FUNCTION "Cage 12 unit" : VOID	// FC 25
TITLE = CAGE 12 UNIT FUNCTION
AUTHOR : Milesi
VERSION : 0.1
VAR_TEMP
  Brake_value : INT ;
END_VAR
BEGIN
NETWORK
TITLE = CAGE 12 OFF
      A(;
      L     "Cage 12".DB25_DBW2;
      L     0;
      ==I;
      );
      AN    "M180.1";
      AN    "M20.0";
      JNB   M001;
      R     "M188.0";
M001: NOP   0;
NETWORK
TITLE = CAGE 12 ON
      A(;
      L     "Cage 12".DB25_DBW2;
      L     1;
      ==I;
      );
      AN    "M180.1";
      AN    "M20.0";
      JNB   M002;
      S     "M188.0";
M002: NOP   0;
NETWORK
TITLE = CAGE 12 Z ROTATION
      A(;
      L     "Cage 12".DB25_DBW4;
      L     0;
      ==I;
      );
      AN    "M180.1";
      AN    "M20.0";
      JNB   M003;
      S     "M188.2";
      R     "M188.3";
M003: NOP   0;
NETWORK
TITLE = CAGE 12 S ROTATION
      A(;
      L     "Cage 12".DB25_DBW4;
      L     1;
      ==I;
      );
      AN    "M180.1";
      AN    "M20.0";
      JNB   M004;
      S     "M188.3";
      R     "M188.2";
M004: NOP   0;
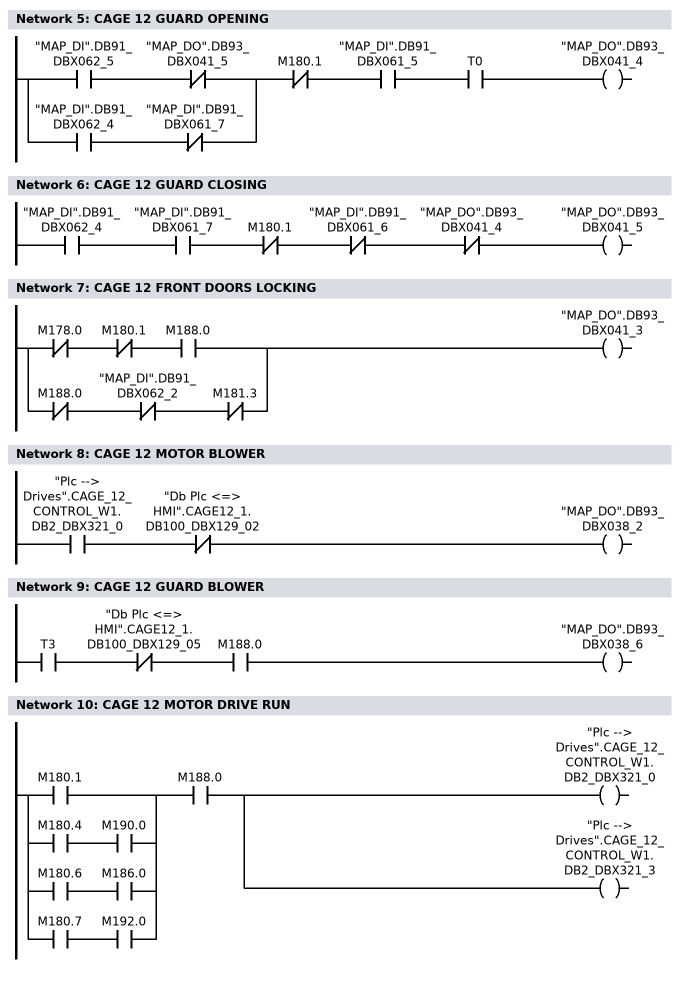
NETWORK
TITLE = CAGE 12 GUARD OPENING
      A(;
      A     "MAP_DI".DB91_DBX062_5;
      AN    "MAP_DO".DB93_DBX041_5;
      O;
      A     "MAP_DI".DB91_DBX062_4;
      AN    "MAP_DI".DB91_DBX061_7;
      );
      AN    "M180.1";
      A     "MAP_DI".DB91_DBX061_5;
      A     "T0";
      =     "MAP_DO".DB93_DBX041_4;
NETWORK
TITLE = CAGE 12 GUARD CLOSING
      A     "MAP_DI".DB91_DBX062_4;
      A     "MAP_DI".DB91_DBX061_7;
//      U     E     66.0
      AN    "M180.1";
      AN    "MAP_DI".DB91_DBX061_6;
      AN    "MAP_DO".DB93_DBX041_4;
      =     "MAP_DO".DB93_DBX041_5;
NETWORK
TITLE = CAGE 12 FRONT DOORS LOCKING
      AN    "M178.0";
      AN    "M180.1";
      A     "M188.0";
      O;
      AN    "M188.0";
      AN    "MAP_DI".DB91_DBX062_2;
      AN    "M181.3";
      =     "MAP_DO".DB93_DBX041_3;
NETWORK
TITLE = CAGE 12 MOTOR BLOWER 
      A     "Plc --> Drives".CAGE_12_CONTROL_W1.DB2_DBX321_0;
      AN    "Db Plc <=> HMI".CAGE12_1.DB100_DBX129_02;
      =     "MAP_DO".DB93_DBX038_2;
NETWORK
TITLE = CAGE 12 GUARD BLOWER
      A     "T3";
      AN    "Db Plc <=> HMI".CAGE12_1.DB100_DBX129_05;
      A     "M188.0";
      =     "MAP_DO".DB93_DBX038_6;
NETWORK
TITLE = CAGE 12 MOTOR DRIVE RUN
      A(;
      O     "M180.1";
      O;
      A     "M180.4";
      A     "M190.0";
      O;
      A     "M180.6";
      A     "M186.0";
      O;
      A     "M180.7";
      A     "M192.0";
      );
      A     "M188.0";
      =     "Plc --> Drives".CAGE_12_CONTROL_W1.DB2_DBX321_0;
      =     "Plc --> Drives".CAGE_12_CONTROL_W1.DB2_DBX321_3;
NETWORK
TITLE = CAGE 12 LAY SET ENABLE
      O     "M180.1";
      O     "M180.5";
      O(;
      A     "M180.4";
      A     "M190.0";
      );
      O(;
      A     "M180.6";
      A     "M186.0";
      );
      O(;
      A     "M180.7";
      A     "M192.0";
      );
      JC    M008;
      L     "Cage 12".DB25_DBD20;
      T     "Cage 12".DB25_DBD24;
      JU    M009;
M008: L     "Cage 12".DB25_DBD24;
      T     "Cage 12".DB25_DBD20;
M009: NOP   0;
NETWORK
TITLE = CAGE 12 MOTOR REFERENCE
//Max Linear Speed = 60 m/min
//Max Cage Rpm = 320
//
//Max Linear Speed              60000
//---------------- = Cage Lay = ----- = 187.5
//  Max Cage Rpm                 320
//
//                             Max Linear Speed
//Max Cage Rpm = 320 = 16384 = ---------------- * K
//                                Cage Lay
//
//    Cage Lay * 16384   187.5 * 16384
//K = ---------------- = ------------- = 51200
//    Max Linear Speed        60
// (network holds code this reader does not know; not shown)
//L     1.121200e+000
NETWORK
TITLE = CAGE 12 MAX LINEAR SPEED TO START
      AN    "M200.1";
      JNB   M00a;
      L     "Cage 12".DB25_DBD24;
      L     2.000000e-01;
      *R;
      JU    M00b;
M00a: L     "Cage 12".DB25_DBD24;
      L     2.600000e-01;
      *R;
M00b: T     "Cage 12".DB25_DBD120;
      O(;
      L     6.000000e+01;
      >R;
      );
      ON    "M188.0";
      JNB   M00c;
      T     "Cage 12".DB25_DBD120;
M00c: NOP   0;
NETWORK
TITLE = CAGE 12 MAX LINEAR SPEED
      L     "Cage 12".DB25_DBD24;
      L     3.200000e-01;
      *R;
      T     "Cage 12".DB25_DBD96;
      O(;
      L     6.000000e+01;
      >R;
      );
      ON    "M188.0";
      JNB   M00d;
      T     "Cage 12".DB25_DBD96;
M00d: NOP   0;
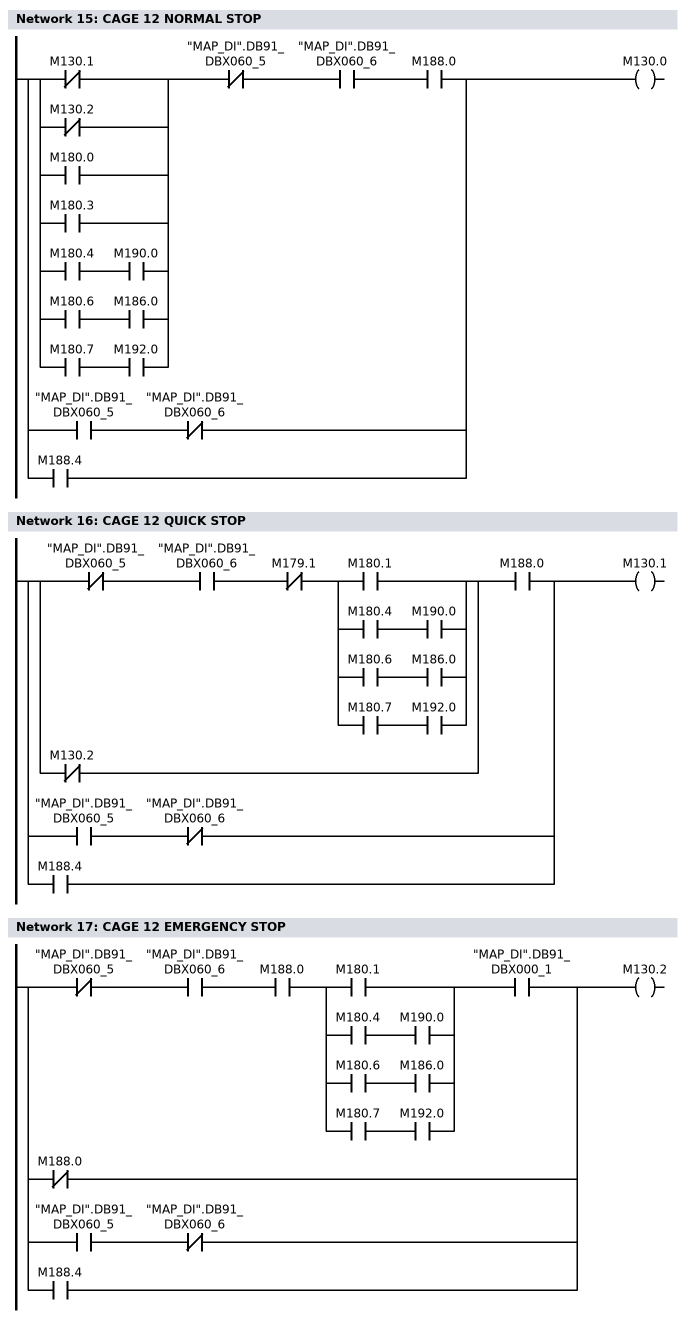
NETWORK
TITLE = CAGE 12 NORMAL STOP
      A(;
      ON    "M130.1";
      ON    "M130.2";
      O     "M180.0";
      O     "M180.3";
      O;
      A     "M180.4";
      A     "M190.0";
      O;
      A     "M180.6";
      A     "M186.0";
      O;
      A     "M180.7";
      A     "M192.0";
      );
      AN    "MAP_DI".DB91_DBX060_5;
      A     "MAP_DI".DB91_DBX060_6;
      A     "M188.0";
      O;
      A     "MAP_DI".DB91_DBX060_5;
      AN    "MAP_DI".DB91_DBX060_6;
      O     "M188.4";
      =     "M130.0";
NETWORK
TITLE = CAGE 12 QUICK STOP
      A(;
      AN    "MAP_DI".DB91_DBX060_5;
      A     "MAP_DI".DB91_DBX060_6;
      AN    "M179.1";
      A(;
      O     "M180.1";
      O;
      A     "M180.4";
      A     "M190.0";
      O;
      A     "M180.6";
      A     "M186.0";
      O;
      A     "M180.7";
      A     "M192.0";
      );
      ON    "M130.2";
      );
      A     "M188.0";
      O;
      A     "MAP_DI".DB91_DBX060_5;
      AN    "MAP_DI".DB91_DBX060_6;
      O     "M188.4";
      =     "M130.1";
NETWORK
TITLE = CAGE 12 EMERGENCY STOP
      AN    "MAP_DI".DB91_DBX060_5;
      A     "MAP_DI".DB91_DBX060_6;
      A     "M188.0";
      A(;
      O     "M180.1";
      O;
      A     "M180.4";
      A     "M190.0";
      O;
      A     "M180.6";
      A     "M186.0";
      O;
      A     "M180.7";
      A     "M192.0";
      );
      A     "MAP_DI".DB91_DBX000_1;
      ON    "M188.0";
      O;
      A     "MAP_DI".DB91_DBX060_5;
      AN    "MAP_DI".DB91_DBX060_6;
      O     "M188.4";
      =     "M130.2";
NETWORK
TITLE = CAGE 12 BRAKE PROPORTIONAL VALVE REFERENCE
      A     "M130.0";
      JC    M005;
      L     "Cage 12".DB25_DBD64;
      L     1.000000e+02;
      /R;
      L     2.764800e+04;
      *R;
      RND;
      JU    M006;
M005: A     "M130.1";
      JC    M007;
      L     "Cage 12".DB25_DBD68;
      L     1.000000e+02;
      /R;
      L     2.764800e+04;
      *R;
      RND;
      JU    M006;
M007: A     "M130.2";
      JC    M011;
      L     "Cage 12".DB25_DBD72;
      L     1.000000e+02;
      /R;
      L     2.764800e+04;
      *R;
      RND;
      JU    M006;
M011: L     0;
M006: T     #Brake_value;
NETWORK
TITLE = SET POINT IN AMPER CALCULATION
      L     "Cage 12".DB20_DBD276;
      L     1.360000e+02;
      *R;
      L     1.000000e+02;
      /R;
      T     "Cage 12".DB20_DBD260;
NETWORK
TITLE = CURRENT CALCULATION
// (network holds code this reader does not know; not shown)
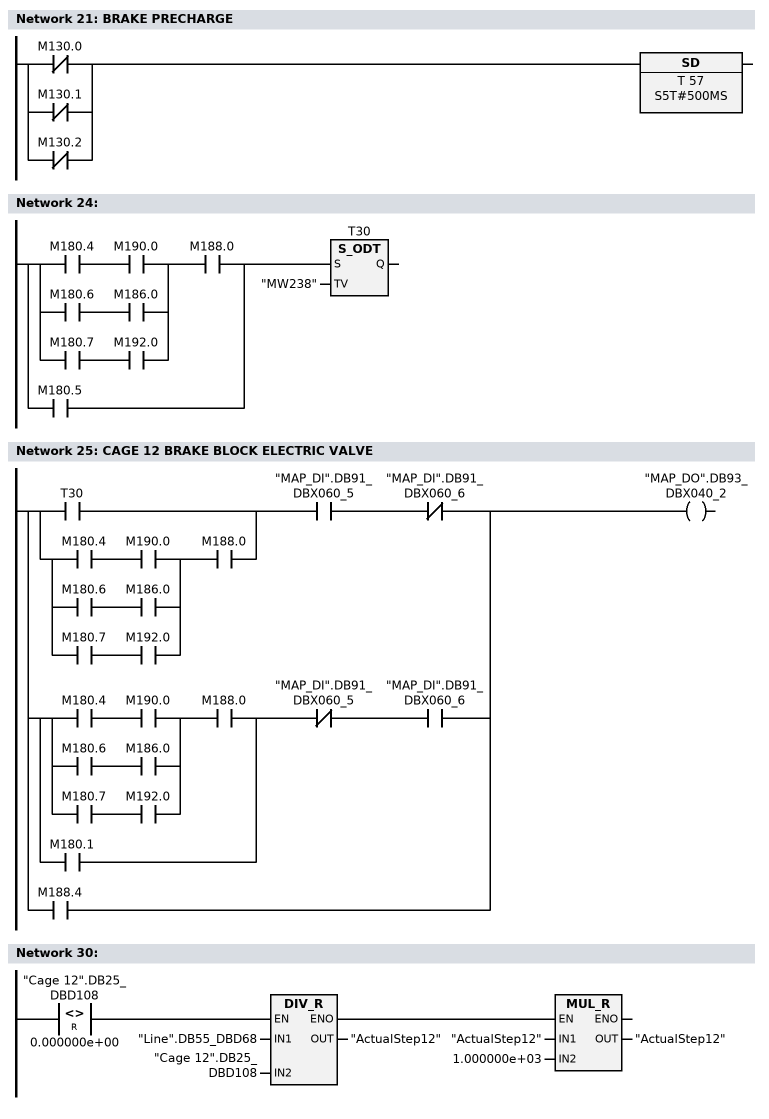
NETWORK
TITLE = BRAKE PRECHARGE
      ON    "M130.0";
      ON    "M130.1";
      ON    "M130.2";
      L     S5T#500MS;
      SD    T 57;
NETWORK
TITLE = BRAKE MODULATION CONTROL
      L     "Cage 12".DB20_DBD260;
      L     "Cage 12".DB25_DBD200;
      -R;
      T     "Cage 12".DB20_DBD264;
      L     "Cage 12".DB20_DBD268;
      *R;
      T     "Cage 12".DB20_DBD272;
      L     2.768400e+04;
      >R;
      JCN   M015;
      L     2.768400e+04;
      T     "Cage 12".DB20_DBD272;
M015: A     T 57;
      A     "M180.1";
      JCN   M016;
      A(;
      L     "Cage 12".DB20_DBD272;
      L     0.000000e+00;
      <R;
      );
      JCN   M017;
      L     0.000000e+00;
      T     "Cage 12".DB20_DBD272;
M017: L     "Cage 12".DB20_DBD272;
      RND;
      JU    M018;
M016: L     #Brake_value;
M018: T     "PAW286";
NETWORK
TITLE = CAGE 12 BRAKE BLOCK OPEN ON-DELAY TIMER
      L     "Cage 12".DB25_DBD148;
      RND;
      ITB;
      L     W#16#2000;
      OW;
      T     "MW238";
NETWORK
TITLE =
      A(;
      A(;
      A     "M180.4";
      A     "M190.0";
      O;
      A     "M180.6";
      A     "M186.0";
      O;
      A     "M180.7";
      A     "M192.0";
      );
      A     "M188.0";
      O     "M180.5";
      );
      L     "MW238";
      SD    "T30";
      NOP   0;
      NOP   0;
      NOP   0;
      NOP   0;
NETWORK
TITLE = CAGE 12 BRAKE BLOCK ELECTRIC VALVE
      A(;
      O     "T30";
      O;
      A(;
      O;
      A     "M180.4";
      A     "M190.0";
      O;
      A     "M180.6";
      A     "M186.0";
      O;
      A     "M180.7";
      A     "M192.0";
      );
      A     "M188.0";
      );
      A     "MAP_DI".DB91_DBX060_5;
      AN    "MAP_DI".DB91_DBX060_6;
      O;
      A(;
      A(;
      O;
      A     "M180.4";
      A     "M190.0";
      O;
      A     "M180.6";
      A     "M186.0";
      O;
      A     "M180.7";
      A     "M192.0";
      );
      A     "M188.0";
      O     "M180.1";
      );
      AN    "MAP_DI".DB91_DBX060_5;
      A     "MAP_DI".DB91_DBX060_6;
      O     "M188.4";
      =     "MAP_DO".DB93_DBX040_2;
NETWORK
TITLE = CAGE 12 RPM TO HMI
      L     "Drives --> Plc".DB1_DBW326;
      ITD;
      DTR;
      L     1.638400e+04;
      /R;
      L     3.200000e+02;
      *R;
      ABS;
      T     "Cage 12".DB25_DBD108;
NETWORK
TITLE = CAGE 12 MOTOR RPM TO HMI
      L     "Drives --> Plc".DB1_DBW326;
      ITD;
      DTR;
      L     1.638400e+04;
      /R;
      L     1.495000e+03;
      *R;
      T     "Cage 12".DB25_DBD188;
NETWORK
TITLE = CAGE 12 MOTOR CURRENT TO HMI
      L     "Drives --> Plc".DB1_DBW328;
      ITD;
      DTR;
      L     1.638400e+04;
      /R;
      L     1.360000e+02;
      *R;
      T     "Cage 12".DB25_DBD192;
NETWORK
TITLE = CAGE 12 MOTOR VOLTAGE TO HMI
      L     "Drives --> Plc".DB1_DBW330;
      ITD;
      DTR;
      L     1.638400e+04;
      /R;
      L     4.000000e+02;
      *R;
      T     "Cage 12".DB25_DBD196;
NETWORK
TITLE =
      A(;
      A(;
      L     "Cage 12".DB25_DBD108;
      L     0.000000e+00;
      <>R;
      );
      JNB   _001;
      L     "Line".DB55_DBD68;
      L     "Cage 12".DB25_DBD108;
      /R;
      T     "ActualStep12";
      AN    OV;
      SAVE;
      CLR;
_001: A     BR;
      );
      JNB   _002;
      L     "ActualStep12";
      L     1.000000e+03;
      *R;
      T     "ActualStep12";
_002: NOP   0;
END_FUNCTION

FUNCTION "Cage 12 loading fase" : VOID	// FC 26
TITLE = CAGE 12 LOADING FASE FUNCTION
AUTHOR : Milesi
VERSION : 0.1
BEGIN
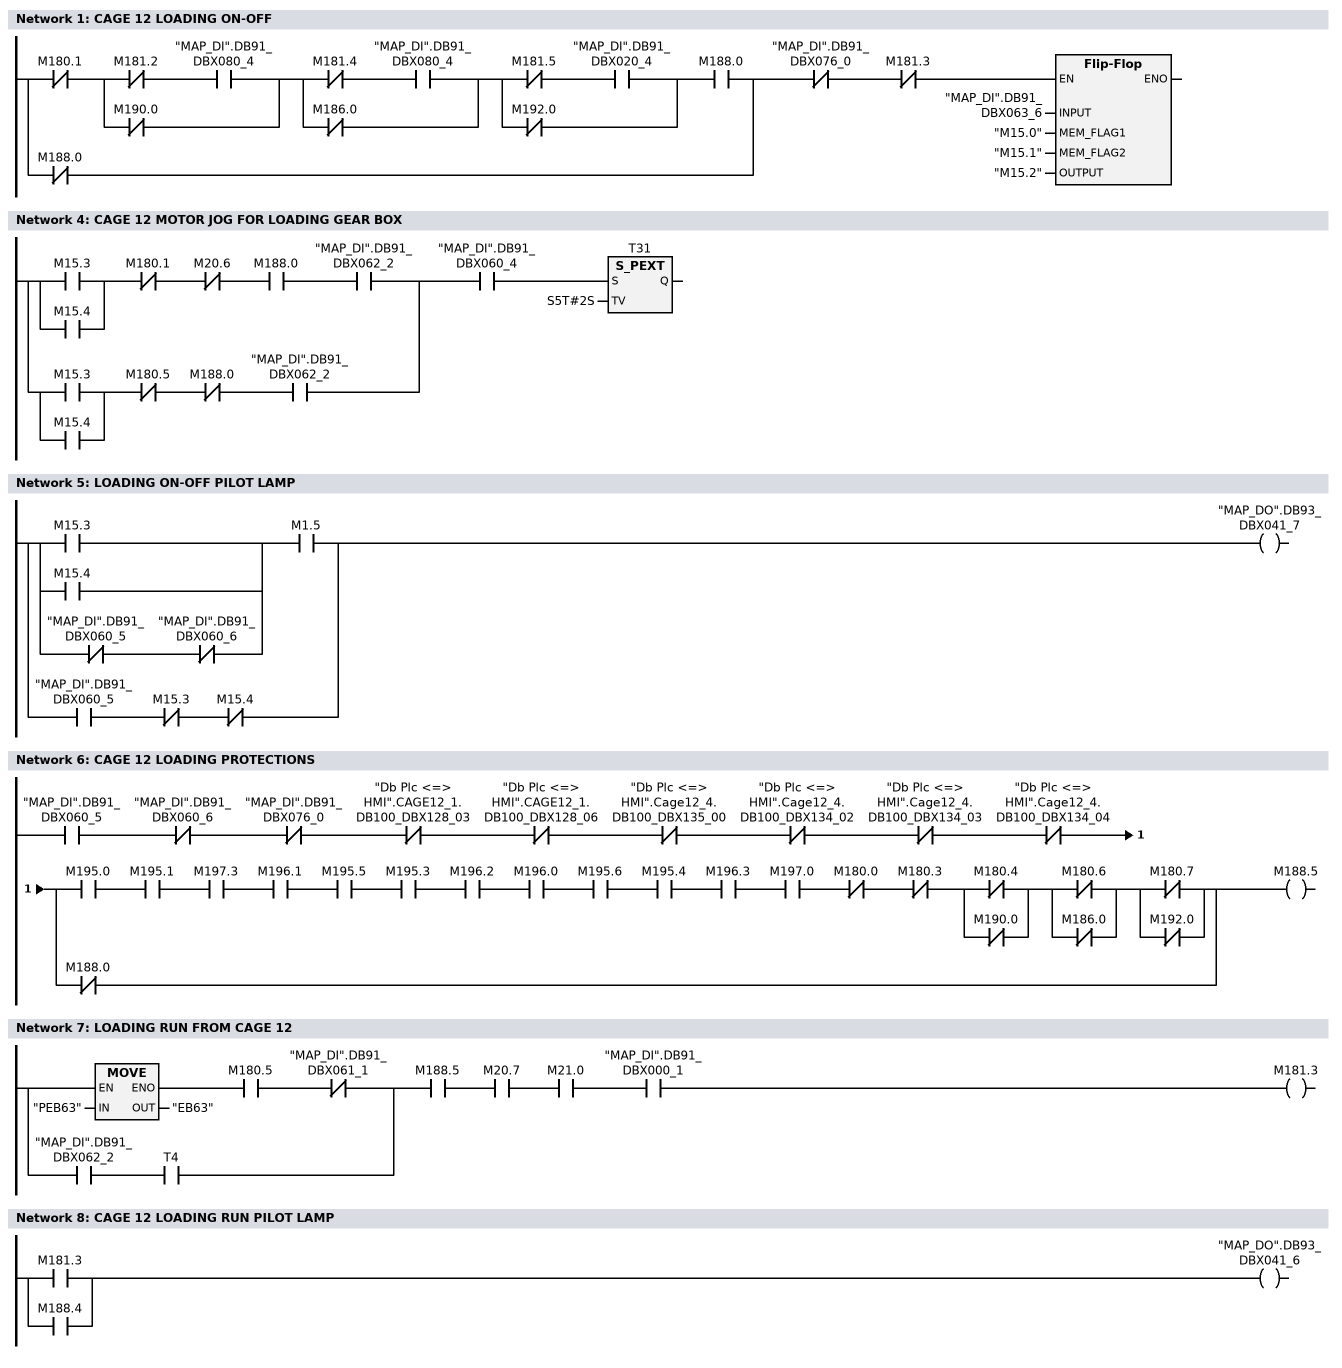
NETWORK
TITLE = CAGE 12 LOADING ON-OFF
      A(;
      AN    "M180.1";
      A(;
      AN    "M181.2";
      A     "MAP_DI".DB91_DBX080_4;
      ON    "M190.0";
      );
      A(;
      AN    "M181.4";
      A     "MAP_DI".DB91_DBX080_4;
      ON    "M186.0";
      );
      A(;
      AN    "M181.5";
      A     "MAP_DI".DB91_DBX020_4;
      ON    "M192.0";
      );
      A     "M188.0";
      ON    "M188.0";
      );
      AN    "MAP_DI".DB91_DBX076_0;
      AN    "M181.3";
      JNB   _001;
      CALL  "Flip-Flop" (
           INPUT                    := "MAP_DI".DB91_DBX063_6,
           MEM_FLAG1                := "M15.0",
           MEM_FLAG2                := "M15.1",
           OUTPUT                   := "M15.2");
_001: NOP   0;
NETWORK
TITLE = CAGE 12 LOADING ON
      A(;
      A(;
      A     "M15.2";
      AN    "M180.1";
      AN    "M20.6";
      A     "M188.0";
      O;
      AN    "M180.5";
      AN    "M188.0";
      );
      S     "MAP_DO".DB93_DBX040_0;
      A(;
      O     "MAP_DI".DB91_DBX060_5;
      O     "MAP_DO".DB93_DBX040_1;
      ON    "M15.2";
      );
      R     "MAP_DO".DB93_DBX040_0;
      A     "MAP_DO".DB93_DBX040_0;
      );
      S     "M15.3";
      A(;
      O     "MAP_DI".DB91_DBX060_5;
      ON    "M15.2";
      );
      R     "M15.3";
      NOP   0;
NETWORK
TITLE = CAGE 12 LOADING OFF
      A(;
      A(;
      AN    "M15.2";
      AN    "M20.6";
      A     "M188.0";
      O;
      AN    "M180.5";
      AN    "M188.0";
      );
      S     "MAP_DO".DB93_DBX040_1;
      A(;
      O     "MAP_DI".DB91_DBX060_6;
      O     "MAP_DO".DB93_DBX040_0;
      O     "M15.2";
      );
      R     "MAP_DO".DB93_DBX040_1;
      A     "MAP_DO".DB93_DBX040_1;
      );
      S     "M15.4";
      A(;
      O     "MAP_DI".DB91_DBX060_6;
      O     "M15.2";
      );
      R     "M15.4";
      NOP   0;
NETWORK
TITLE = CAGE 12 MOTOR JOG FOR LOADING GEAR BOX
      A(;
      A(;
      O     "M15.3";
      O     "M15.4";
      );
      AN    "M180.1";
      AN    "M20.6";
      A     "M188.0";
      A     "MAP_DI".DB91_DBX062_2;
      O;
      A(;
      O     "M15.3";
      O     "M15.4";
      );
      AN    "M180.5";
      AN    "M188.0";
      A     "MAP_DI".DB91_DBX062_2;
      );
      A     "MAP_DI".DB91_DBX060_4;
      L     S5T#2S;
      SE    "T31";
      NOP   0;
      NOP   0;
      NOP   0;
      NOP   0;
NETWORK
TITLE = LOADING ON-OFF PILOT LAMP
      A(;
      O     "M15.3";
      O     "M15.4";
      O;
      AN    "MAP_DI".DB91_DBX060_5;
      AN    "MAP_DI".DB91_DBX060_6;
      );
      A     "M1.5";
      O;
      A     "MAP_DI".DB91_DBX060_5;
      AN    "M15.3";
      AN    "M15.4";
      =     "MAP_DO".DB93_DBX041_7;
NETWORK
TITLE = CAGE 12 LOADING PROTECTIONS
      A     "MAP_DI".DB91_DBX060_5;
      AN    "MAP_DI".DB91_DBX060_6;
      AN    "MAP_DI".DB91_DBX076_0;
      AN    "Db Plc <=> HMI".CAGE12_1.DB100_DBX128_03;
      AN    "Db Plc <=> HMI".CAGE12_1.DB100_DBX128_06;
      AN    "Db Plc <=> HMI".Cage12_4.DB100_DBX135_00;
      AN    "Db Plc <=> HMI".Cage12_4.DB100_DBX134_02;
      AN    "Db Plc <=> HMI".Cage12_4.DB100_DBX134_03;
      AN    "Db Plc <=> HMI".Cage12_4.DB100_DBX134_04;
      A(;
      A     "M195.0";
      A     "M195.1";
      A     "M197.3";
      A     "M196.1";
      A     "M195.5";
      A     "M195.3";
      A     "M196.2";
      A     "M196.0";
      A     "M195.6";
      A     "M195.4";
      A     "M196.3";
      A     "M197.0";
      AN    "M180.0";
      AN    "M180.3";
      A(;
      ON    "M180.4";
      ON    "M190.0";
      );
      A(;
      ON    "M180.6";
      ON    "M186.0";
      );
      A(;
      ON    "M180.7";
      ON    "M192.0";
      );
      ON    "M188.0";
      );
      =     "M188.5";
NETWORK
TITLE = LOADING RUN FROM CAGE 12
      A(;
      A(;
      L     "PEB63";
      T     "EB63";
      SET;
      SAVE;
      CLR;
      A     BR;
      );
      A     "M180.5";
      AN    "MAP_DI".DB91_DBX061_1;
      O;
      A     "MAP_DI".DB91_DBX062_2;
      A     "T4";
      );
      A     "M188.5";
      A     "M20.7";
      A     "M21.0";
      A     "MAP_DI".DB91_DBX000_1;
      =     "M181.3";
NETWORK
TITLE = CAGE 12 LOADING RUN PILOT LAMP
      O     "M181.3";
      O     "M188.4";
      =     "MAP_DO".DB93_DBX041_6;
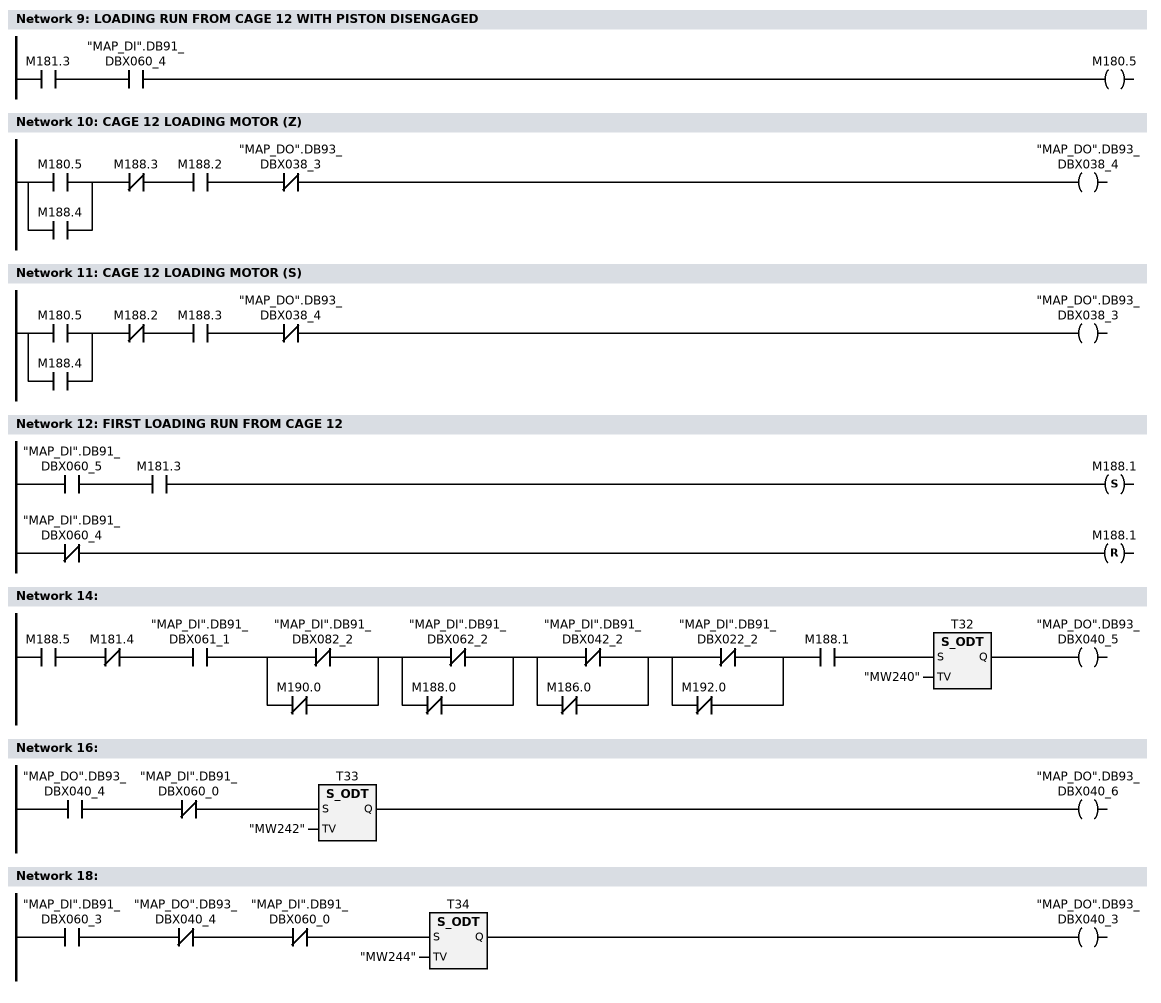
NETWORK
TITLE = LOADING RUN FROM CAGE 12 WITH PISTON DISENGAGED
      A     "M181.3";
      A     "MAP_DI".DB91_DBX060_4;
      =     "M180.5";
NETWORK
TITLE = CAGE 12 LOADING MOTOR (Z)
      A(;
      O     "M180.5";
      O     "M188.4";
      );
      AN    "M188.3";
      A     "M188.2";
      AN    "MAP_DO".DB93_DBX038_3;
      =     "MAP_DO".DB93_DBX038_4;
NETWORK
TITLE = CAGE 12 LOADING MOTOR (S)
      A(;
      O     "M180.5";
      O     "M188.4";
      );
      AN    "M188.2";
      A     "M188.3";
      AN    "MAP_DO".DB93_DBX038_4;
      =     "MAP_DO".DB93_DBX038_3;
NETWORK
TITLE = FIRST LOADING RUN FROM CAGE 12
      A     "MAP_DI".DB91_DBX060_5;
      A     "M181.3";
      S     "M188.1";
      AN    "MAP_DI".DB91_DBX060_4;
      R     "M188.1";
      NOP   0;
NETWORK
TITLE = CAGE 12 PISTON ENGAGING INTO CAGE
      L     "Cage 12".DB25_DBD152;
      RND;
      ITB;
      L     W#16#2000;
      OW;
      T     "MW240";
NETWORK
TITLE =
      A     "M188.5";
      AN    "M181.4";
      A     "MAP_DI".DB91_DBX061_1;
      A(;
      ON    "MAP_DI".DB91_DBX082_2;
      ON    "M190.0";
      );
      A(;
      ON    "MAP_DI".DB91_DBX062_2;
      ON    "M188.0";
      );
      A(;
      ON    "MAP_DI".DB91_DBX042_2;
      ON    "M186.0";
      );
      A(;
      ON    "MAP_DI".DB91_DBX022_2;
      ON    "M192.0";
      );
      A     "M188.1";
      L     "MW240";
      SD    "T32";
      NOP   0;
      NOP   0;
      NOP   0;
      A     "T32";
      =     "MAP_DO".DB93_DBX040_5;
NETWORK
TITLE = CAGE 12 PISTON DISENGAGING FROM CAGE
      L     "Cage 12".DB25_DBD144;
      RND;
      ITB;
      L     W#16#2000;
      OW;
      T     "MW242";
NETWORK
TITLE =
      A     "MAP_DO".DB93_DBX040_4;
      AN    "MAP_DI".DB91_DBX060_0;
      L     "MW242";
      SD    "T33";
      NOP   0;
      NOP   0;
      NOP   0;
      A     "T33";
      =     "MAP_DO".DB93_DBX040_6;
NETWORK
TITLE = CAGE 12 AIR INLET INTO CAGE
      L     "Cage 12".DB25_DBD156;
      RND;
      ITB;
      L     W#16#2000;
      OW;
      T     "MW244";
NETWORK
TITLE =
      A     "MAP_DI".DB91_DBX060_3;
      AN    "MAP_DO".DB93_DBX040_4;
      AN    "MAP_DI".DB91_DBX060_0;
      L     "MW244";
      SD    "T34";
      NOP   0;
      NOP   0;
      NOP   0;
      A     "T34";
      =     "MAP_DO".DB93_DBX040_3;
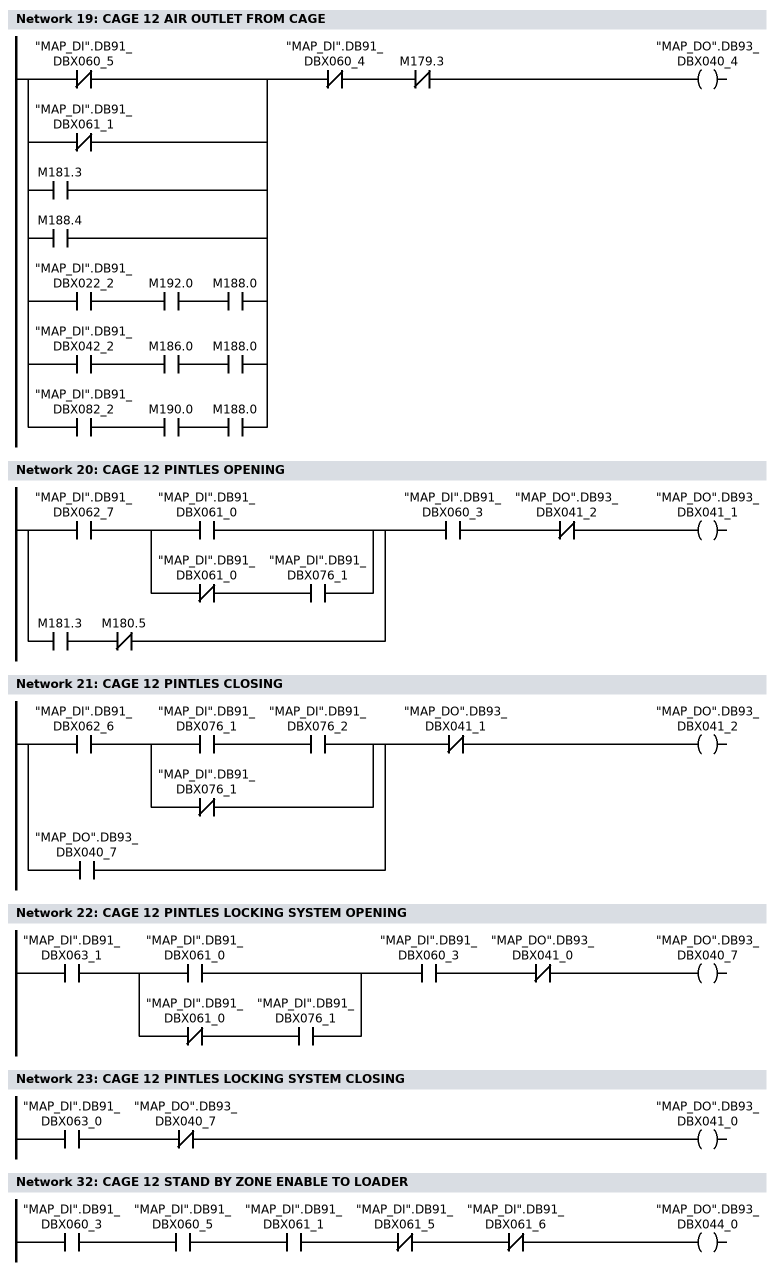
NETWORK
TITLE = CAGE 12 AIR OUTLET FROM CAGE
      A(;
      ON    "MAP_DI".DB91_DBX060_5;
      ON    "MAP_DI".DB91_DBX061_1;
      O     "M181.3";
      O     "M188.4";
      O;
      A     "MAP_DI".DB91_DBX022_2;
      A     "M192.0";
      A     "M188.0";
      O;
      A     "MAP_DI".DB91_DBX042_2;
      A     "M186.0";
      A     "M188.0";
      O;
      A     "MAP_DI".DB91_DBX082_2;
      A     "M190.0";
      A     "M188.0";
      );
      AN    "MAP_DI".DB91_DBX060_4;
      AN    "M179.3";
      =     "MAP_DO".DB93_DBX040_4;
NETWORK
TITLE = CAGE 12 PINTLES OPENING
      A(;
      A     "MAP_DI".DB91_DBX062_7;
      A(;
      O     "MAP_DI".DB91_DBX061_0;
      O;
      AN    "MAP_DI".DB91_DBX061_0;
      A     "MAP_DI".DB91_DBX076_1;
      );
      O;
      A     "M181.3";
      AN    "M180.5";
      );
      A     "MAP_DI".DB91_DBX060_3;
      AN    "MAP_DO".DB93_DBX041_2;
      =     "MAP_DO".DB93_DBX041_1;
NETWORK
TITLE = CAGE 12 PINTLES CLOSING
      A(;
      A     "MAP_DI".DB91_DBX062_6;
      A(;
      A     "MAP_DI".DB91_DBX076_1;
      A     "MAP_DI".DB91_DBX076_2;
      ON    "MAP_DI".DB91_DBX076_1;
      );
      O     "MAP_DO".DB93_DBX040_7;
      );
      AN    "MAP_DO".DB93_DBX041_1;
      =     "MAP_DO".DB93_DBX041_2;
NETWORK
TITLE = CAGE 12 PINTLES LOCKING SYSTEM OPENING
      A     "MAP_DI".DB91_DBX063_1;
      A(;
      O     "MAP_DI".DB91_DBX061_0;
      O;
      AN    "MAP_DI".DB91_DBX061_0;
      A     "MAP_DI".DB91_DBX076_1;
      );
      A     "MAP_DI".DB91_DBX060_3;
      AN    "MAP_DO".DB93_DBX041_0;
      =     "MAP_DO".DB93_DBX040_7;
NETWORK
TITLE = CAGE 12 PINTLES LOCKING SYSTEM CLOSING
      A     "MAP_DI".DB91_DBX063_0;
      AN    "MAP_DO".DB93_DBX040_7;
      =     "MAP_DO".DB93_DBX041_0;
NETWORK
TITLE = CAGE 12 PLATFORM UP
NETWORK
TITLE = CAGE 12 PLATFORM DOWN
NETWORK
TITLE = CAGE 12 EVEN BOBBINS ROTATION FOR LOADING MACHINE
NETWORK
TITLE = CAGE 12 EVEN BOBBINS ROTATION FOR LOADING PLATFORM
NETWORK
TITLE = CAGE 12 ODD BOBBINS ROTATION FOR LOADING MACHINE
NETWORK
TITLE = CAGE 12 ODD BOBBINS ROTATION FOR LOADING PLATFORM
NETWORK
TITLE = CAGE 12 BOBBIN ROTATION FOR LOADING MACHINE PILOT LAMP
NETWORK
TITLE = CAGE 12 LOADING PUMP
NETWORK
TITLE = CAGE 12 STAND BY ZONE ENABLE TO LOADER
      A     "MAP_DI".DB91_DBX060_3;
      A     "MAP_DI".DB91_DBX060_5;
      A     "MAP_DI".DB91_DBX061_1;
      AN    "MAP_DI".DB91_DBX061_5;
      AN    "MAP_DI".DB91_DBX061_6;
      =     "MAP_DO".DB93_DBX044_0;
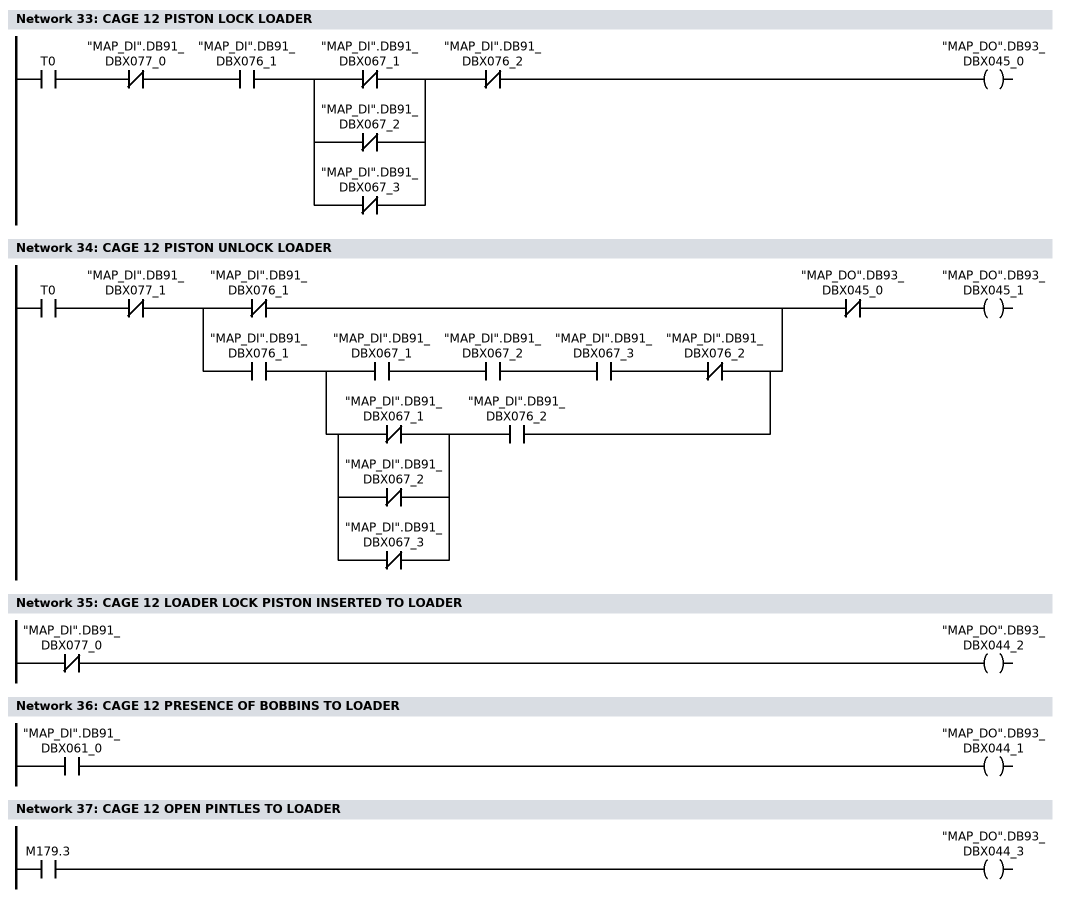
NETWORK
TITLE = CAGE 12 PISTON LOCK LOADER
      A     "T0";
      AN    "MAP_DI".DB91_DBX077_0;
      A     "MAP_DI".DB91_DBX076_1;
      A(;
      ON    "MAP_DI".DB91_DBX067_1;
      ON    "MAP_DI".DB91_DBX067_2;
      ON    "MAP_DI".DB91_DBX067_3;
      );
      AN    "MAP_DI".DB91_DBX076_2;
      =     "MAP_DO".DB93_DBX045_0;
NETWORK
TITLE = CAGE 12 PISTON UNLOCK LOADER
      A     "T0";
      AN    "MAP_DI".DB91_DBX077_1;
      A(;
      ON    "MAP_DI".DB91_DBX076_1;
      O;
      A     "MAP_DI".DB91_DBX076_1;
      A(;
      A     "MAP_DI".DB91_DBX067_1;
      A     "MAP_DI".DB91_DBX067_2;
      A     "MAP_DI".DB91_DBX067_3;
      AN    "MAP_DI".DB91_DBX076_2;
      O;
      A(;
      ON    "MAP_DI".DB91_DBX067_1;
      ON    "MAP_DI".DB91_DBX067_2;
      ON    "MAP_DI".DB91_DBX067_3;
      );
      A     "MAP_DI".DB91_DBX076_2;
      );
      );
      AN    "MAP_DO".DB93_DBX045_0;
      =     "MAP_DO".DB93_DBX045_1;
NETWORK
TITLE = CAGE 12 LOADER LOCK PISTON INSERTED TO LOADER 
      AN    "MAP_DI".DB91_DBX077_0;
      =     "MAP_DO".DB93_DBX044_2;
NETWORK
TITLE = CAGE 12 PRESENCE OF BOBBINS TO LOADER
      A     "MAP_DI".DB91_DBX061_0;
      =     "MAP_DO".DB93_DBX044_1;
NETWORK
TITLE = CAGE 12 OPEN PINTLES TO LOADER
      A     "M179.3";
      =     "MAP_DO".DB93_DBX044_3;
END_FUNCTION

FUNCTION "Cage 12 preforming alarm" : VOID	// FC 27
TITLE = CAGE 12 PREFORMING ALARMS FUNCTION
AUTHOR : Milesi
VERSION : 0.1
BEGIN
NETWORK
TITLE = CAGE 12 PREFORMING MOTOR DRIVE PROFIBUS SLAVE 10 FAULT
      A(;
      L     "MB304";
      L     10;
      ==I;
      );
      AN    "M300.5";
      S     "Db Plc <=> HMI".PROFIBUS.DB100_DBX100_1;
NETWORK
TITLE = CAGE 12 PREFORMING MOTOR BRAKE OVERLOAD
      A     "T0";
      A     "MAP_DI".DB91_DBX058_4;
      A     "M189.3";
      =     "Db Plc <=> HMI".Cage12_4.DB100_DBX135_04;
NETWORK
TITLE = CAGE 12 PREFORMING MOTOR BLOWER OVERLOAD
      A     "T0";
      A     "MAP_DI".DB91_DBX058_5;
      A     "M189.3";
      =     "Db Plc <=> HMI".Cage12_4.DB100_DBX135_05;
NETWORK
TITLE = CAGE 12 PREFORMING OPEN GUARD
      A     "T0";
      A     "M180.1";
      AN    "MAP_DI".DB91_DBX064_6;
      A     "M189.3";
      S     "M174.5";
NETWORK
TITLE =
      A     "T0";
      A(;
      ON    "MAP_DI".DB91_DBX064_6;
      O     "M174.5";
      );
      A     "M189.3";
      =     "Db Plc <=> HMI".Cage12_4.DB100_DBX135_06;
NETWORK
TITLE = CAGE 12 PREFORMING MOTOR DRIVE FAULT
      A     "T0";
      A     "Drives --> Plc".CAGE_12_PREF_STATUS_W1.DB1_DBX281_3;
      A     "M189.3";
      S     "Db Plc <=> HMI".Cage12_4.DB100_DBX135_07;
NETWORK
TITLE = CAGE 12 PREFORMING GENERAL ALARM
      AN    "Db Plc <=> HMI".PROFIBUS.DB100_DBX100_1;
      AN    "Db Plc <=> HMI".Cage12_4.DB100_DBX135_04;
      AN    "Db Plc <=> HMI".Cage12_4.DB100_DBX135_05;
      AN    "Db Plc <=> HMI".Cage12_4.DB100_DBX135_06;
      AN    "Db Plc <=> HMI".Cage12_4.DB100_DBX135_07;
      =     "M196.0";
END_FUNCTION

FUNCTION "Cage 12 preforming unit" : VOID	// FC 28
TITLE = CAGE 12 PREFORMING UNIT FUNCTION
AUTHOR : Milesi
VERSION : 0.1
BEGIN
NETWORK
TITLE = CAGE 12 PREFORMING OFF
      A(;
      L     "Cage 12 preforming".DB28_DBW2;
      L     0;
      ==I;
      );
      AN    "M180.1";
      JNB   _001;
      R     "M189.3";
      R     "M189.4";
      R     "M189.5";
_001: NOP   0;
NETWORK
TITLE = CAGE 12 PREFORMING Z ROTATION
      A(;
      L     "Cage 12 preforming".DB28_DBW2;
      L     1;
      ==I;
      );
      AN    "M180.1";
      JNB   _002;
      S     "M189.3";
      S     "M189.4";
      R     "M189.5";
_002: NOP   0;
NETWORK
TITLE = CAGE 12 PREFORMING S ROTATION
      A(;
      L     "Cage 12 preforming".DB28_DBW2;
      L     2;
      ==I;
      );
      AN    "M180.1";
      JNB   _003;
      S     "M189.3";
      S     "M189.5";
      R     "M189.4";
_003: NOP   0;
NETWORK
TITLE = CAGE 12 PREFORMING MOTOR DRIVE RUN
      A(;
      O     "M180.1";
      O     "M21.3";
      );
      AN    "Db Plc <=> HMI".Cage12_4.DB100_DBX135_07;
      A     "M189.3";
      =     "Plc --> Drives".CAGE_12_PREF_CONTROL_W1.DB2_DBX281_0;
      =     "Plc --> Drives".CAGE_12_PREF_CONTROL_W1.DB2_DBX281_3;
NETWORK
TITLE = CAGE 12 PREFORMING MOTOR BLOWER
      A     "Plc --> Drives".CAGE_12_PREF_CONTROL_W1.DB2_DBX281_0;
      AN    "Db Plc <=> HMI".Cage12_4.DB100_DBX135_05;
      =     "MAP_DO".DB93_DBX038_1;
NETWORK
TITLE = CAGE 12 PREFORMING MOTOR ELECTRIC BRAKE RELAY
      A(;
      O     "Plc --> Drives".CAGE_12_PREF_CONTROL_W1.DB2_DBX281_0;
      O     "MAP_DI".DB91_DBX064_7;
      );
      AN    "Db Plc <=> HMI".Cage12_4.DB100_DBX135_05;
      =     "MAP_DO".DB93_DBX038_0;
NETWORK
TITLE = CAGE 12 PREFORMING MOTOR REFERENCE
//Max Linear Speed = 40 m/min
//Max Die Rpm = 147.68
//
//Max Linear Speed             40000
//---------------- = Die Lay = ------ = 270.85
//  Max Die Rpm                147.68
//
//                               Max Linear Speed
//Max Die Rpm = 147.68 = 16384 = ---------------- * K
//                                   Die Lay
//
//    Die Lay * 16384   270.85 * 16384
//K = ---------------- = ------------- = 110940.16
//    Max Linear Speed        40
// (network holds code this reader does not know; not shown)
NETWORK
TITLE = CAGE 12 PREFORMING RPM TO HMI
      L     "Drives --> Plc".DB1_DBW286;
      ITD;
      DTR;
      L     1.638400e+04;
      /R;
      L     1.476800e+02;
      *R;
      ABS;
      T     "Cage 12 preforming".DB28_DBD108;
NETWORK
TITLE = CAGE 12 PREFORMING MOTOR RPM TO HMI
      L     "Drives --> Plc".DB1_DBW286;
      ITD;
      DTR;
      L     1.638400e+04;
      /R;
      L     1.420000e+03;
      *R;
      T     "Cage 12 preforming".DB28_DBD188;
NETWORK
TITLE = CAGE 12 PREFORMING MOTOR CURRENT TO HMI
//TORQUE FEEDBACK = 150% = MOTOR CURRENT * 1.5
      L     "Drives --> Plc".DB1_DBW288;
      ITD;
      DTR;
      L     1.638400e+04;
      /R;
      L     3.400000e+00;
      *R;
      T     "Cage 12 preforming".DB28_DBD192;
NETWORK
TITLE = CAGE 12 PREFORMING MOTOR VOLTAGE TO HMI
      L     "Drives --> Plc".DB1_DBW290;
      ITD;
      DTR;
      L     1.638400e+04;
      /R;
      L     4.000000e+02;
      *R;
      T     "Cage 12 preforming".DB28_DBD196;
END_FUNCTION

FUNCTION "Cage 6 alarms" : VOID	// FC 29
TITLE = CAGE 6 ALARMS FUNCTION
AUTHOR : Milesi
VERSION : 0.1
VAR_TEMP
  T4_time : WORD ;
END_VAR
BEGIN
NETWORK
TITLE = CAGE 6 MOTOR DRIVE PROFIBUS SLAVE 12 FAULT
      A(;
      L     "MB304";
      L     12;
      ==I;
      );
      AN    "M300.5";
      S     "Db Plc <=> HMI".PROFIBUS.DB100_DBX100_3;
NETWORK
TITLE = CAGE 6 ET200M PROFIBUS SLAVE 24 FAULT
      A(;
      L     "MB304";
      L     24;
      ==I;
      );
      AN    "M300.5";
      S     "Db Plc <=> HMI".PROFIBUS_1.DB100_DBX103_0;
NETWORK
TITLE = CAGE 6 OPEN FRONT GUARD
      A     "T0";
      A     "M180.1";
      AN    "MAP_DI".DB91_DBX081_6;
      A     "M190.0";
      S     "M173.1";
NETWORK
TITLE =
      A     "T0";
      A(;
      ON    "MAP_DI".DB91_DBX081_6;
      O     "M173.1";
      );
      A     "M190.0";
      =     "Db Plc <=> HMI".Cage6_1.DB100_DBX136_0;
NETWORK
TITLE = CAGE 6 PRESENCE OF MAN
      A     "T0";
      AN    "MAP_DI".DB91_DBX081_7;
      AN    "M180.1";
      A     "M190.0";
      =     "Db Plc <=> HMI".Cage6_1.DB100_DBX136_1;
NETWORK
TITLE = CAGE 6 LOADING ENGAGED
      A     "T0";
      A     "MAP_DI".DB91_DBX080_5;
      AN    "MAP_DI".DB91_DBX080_6;
      A     "M14.2";
      =     "Db Plc <=> HMI".Cage6_1.DB100_DBX136_2;
NETWORK
TITLE = CAGE 6 LOADING GEAR BOX NOT ENGAGED
      A     "T0";
      AN    "MAP_DI".DB91_DBX080_5;
      AN    "MAP_DI".DB91_DBX080_6;
      =     "Db Plc <=> HMI".Cage6_1.DB100_DBX136_3;
NETWORK
TITLE = CAGE 6 LOADING MOTOR OVERLOAD
      A     "T0";
      A     "MAP_DI".DB91_DBX078_4;
      =     "Db Plc <=> HMI".Cage6_1.DB100_DBX136_6;
NETWORK
TITLE = CAGE 6 AIR PIPE NOT IN POSITION
      A     "T0";
      A     "M180.1";
      AN    "MAP_DI".DB91_DBX080_7;
      A     "M190.0";
      S     "M173.2";
NETWORK
TITLE =
      A     "T0";
      A(;
      ON    "MAP_DI".DB91_DBX080_7;
      O     "M173.2";
      );
      =     "Db Plc <=> HMI".Cage6_1.DB100_DBX136_5;
NETWORK
TITLE = CAGE 6 PISTON INSIDE CAGE
      A     "T0";
      A     "M180.1";
      AN    "MAP_DI".DB91_DBX080_4;
      A     "M190.0";
      S     "M171.5";
NETWORK
TITLE =
      A     "T0";
      A(;
      ON    "MAP_DI".DB91_DBX080_4;
      O     "M171.5";
      );
      =     "Db Plc <=> HMI".Cage6_1.DB100_DBX136_7;
NETWORK
TITLE = CAGE 6 24VDC POWER SUPPLY OVERLOAD
      A     "T0";
      AN    "MAP_DI".DB91_DBX078_3;
      =     "Db Plc <=> HMI".Cage6_1.DB100_DBX137_0;
NETWORK
TITLE = CAGE 6 220VAC POWER SUPPLY OVERLOAD
      A     "T0";
      AN    "MAP_DI".DB91_DBX078_2;
      =     "Db Plc <=> HMI".Cage6_1.DB100_DBX137_1;
NETWORK
TITLE = CAGE 6 MOTOR BLOWER OVERLOAD
      A     "T0";
      A     "MAP_DI".DB91_DBX078_5;
      =     "Db Plc <=> HMI".Cage6_1.DB100_DBX137_2;
NETWORK
TITLE = CAGE 6 LOADING PLATFORM MOTOR OVERLOAD
NETWORK
TITLE = CAGE 6 GUARD BLOWER MOTOR OVERLOAD
      A     "T0";
      A     "MAP_DI".DB91_DBX078_7;
      =     "Db Plc <=> HMI".Cage6_1.DB100_DBX137_5;
NETWORK
TITLE = CAGE 6 OPEN FRONT DOOR
//      U(    
//      U(    
//      U     T      0
//      U     M    178.0
//      O     M    180.1
//      O     M     21.3
//      )     
//      L     S5T#2S
//      SE    T     45
//      NOP   0
//      NOP   0
//      NOP   0
//      U     T     45
//      )     
//      UN    DB91.DBX   81.3
//      U     M    190.0
//      S     DB100.DBX  137.6
NETWORK
TITLE = CAGE 6 OPEN REAR DOORS
      A     "T0";
      A     "M180.1";
      AN    "MAP_DI".DB91_DBX081_4;
      A     "M190.0";
      S     "M172.7";
NETWORK
TITLE =
      A     "T0";
      A(;
      ON    "MAP_DI".DB91_DBX081_4;
      O     "M172.7";
      );
      A     "M190.0";
      =     "Db Plc <=> HMI".Cage6_1.DB100_DBX137_7;
NETWORK
TITLE = CAGE 6 BREAK WIRE FROM RING 
      A     "T0";
      A     "T1";
      AN    "MAP_DI".DB91_DBX081_2;
      A     "M190.0";
      S     "Db Plc <=> HMI".Cage6_3.DB100_DBX141_6;
NETWORK
TITLE = CAGE 6 MAIN AIR MINIMUM PRESSURE
      A     "T0";
      A     "M180.1";
      AN    "MAP_DI".DB91_DBX080_2;
      A     "M190.0";
      S     "M172.4";
NETWORK
TITLE =
      A     "T0";
      A(;
      ON    "MAP_DI".DB91_DBX080_2;
      O     "M172.4";
      );
      =     "Db Plc <=> HMI".Cage6_4.DB100_DBX142_0;
NETWORK
TITLE = CAGE 6 BOBBIN BRAKES AIR TANK MINIMUM PRESSURE
      A     "T0";
      AN    "Db Plc <=> HMI".PROFIBUS_1.DB100_DBX103_0;
      AN    "MAP_DI".DB91_DBX087_0;
      A     "M190.0";
      S     "Db Plc <=> HMI".Cage6_4.DB100_DBX142_1;
NETWORK
TITLE = CAGE 6 LINE 1 PINTLES OPEN
      A     "T0";
      A     "M180.1";
      AN    "MAP_DI".DB91_DBX087_1;
      A     "M190.0";
      S     "M171.6";
NETWORK
TITLE =
      A     "T0";
      A(;
      ON    "MAP_DI".DB91_DBX087_1;
      O     "M171.6";
      );
      =     "Db Plc <=> HMI".Cage6_4.DB100_DBX142_2;
NETWORK
TITLE = CAGE 6 LINE 2 PINTLES OPEN
      A     "T0";
      A     "M180.1";
      AN    "MAP_DI".DB91_DBX087_2;
      A     "M190.0";
      S     "M171.7";
NETWORK
TITLE =
      A     "T0";
      A(;
      ON    "MAP_DI".DB91_DBX087_2;
      O     "M171.7";
      );
      =     "Db Plc <=> HMI".Cage6_4.DB100_DBX142_3;
NETWORK
TITLE = CAGE 6 LINE 3 PINTLES OPEN
      A     "T0";
      A     "M180.1";
      AN    "MAP_DI".DB91_DBX087_3;
      A     "M190.0";
      S     "M172.0";
NETWORK
TITLE =
      A     "T0";
      A(;
      ON    "MAP_DI".DB91_DBX087_3;
      O     "M172.0";
      );
      =     "Db Plc <=> HMI".Cage6_4.DB100_DBX142_4;
NETWORK
TITLE = CAGE 6 OPEN PINTLES LAMP
      ON    "MAP_DI".DB91_DBX087_1;
      ON    "MAP_DI".DB91_DBX087_2;
      ON    "MAP_DI".DB91_DBX087_3;
      =     "M179.2";
      =     "MAP_DO".DB93_DBX052_0;
NETWORK
TITLE = CAGE 6 MOTOR DRIVE FAULT
      A     "T0";
      A     "Drives --> Plc".CAGE_6_STATUS_W1.DB1_DBX361_3;
      S     "Db Plc <=> HMI".Cage6_4.DB100_DBX142_5;
NETWORK
TITLE = CAGE 6 MOTOR OVERTEMPERATURE
      A     "T0";
      A     "Drives --> Plc".CAGE_6_STATUS_W2.DB1_DBX362_1;
      S     "Db Plc <=> HMI".Cage6_4.DB100_DBX142_6;
NETWORK
TITLE = CAGE 6 OVERSPEED
      A     "T0";
      A     "M180.1";
      A(;
      L     "Cage 6".DB30_DBD108;
      L     3.250000e+02;
      >=R;
      );
      A     "M190.0";
      S     "Db Plc <=> HMI".Cage6_4.DB100_DBX142_7;
NETWORK
TITLE = CAGE 6 BRAKES CONTROL
      A     "T0";
      A     "T2";
      AN    "MAP_DI".DB91_DBX080_1;
      A     "M190.0";
      S     "Db Plc <=> HMI".Cage6_4.DB100_DBX143_0;
NETWORK
TITLE = CAGE 6 PLATFORM UP
NETWORK
TITLE = CAGE 6 HYDRAULIC UNIT MINIMUM OIL LEVEL  
NETWORK
TITLE = CAGE 6 GENERAL ALARM
      AN    "Db Plc <=> HMI".PROFIBUS.DB100_DBX100_3;
      AN    "Db Plc <=> HMI".PROFIBUS_1.DB100_DBX103_0;
      AN    "Db Plc <=> HMI".Cage6_1.DB100_DBX136_0;
      AN    "Db Plc <=> HMI".Cage6_1.DB100_DBX136_1;
      AN    "Db Plc <=> HMI".Cage6_1.DB100_DBX136_3;
      AN    "Db Plc <=> HMI".Cage6_1.DB100_DBX136_4;
      AN    "Db Plc <=> HMI".Cage6_1.DB100_DBX136_5;
      AN    "Db Plc <=> HMI".Cage6_1.DB100_DBX136_7;
      AN    "Db Plc <=> HMI".Cage6_1.DB100_DBX137_0;
      AN    "Db Plc <=> HMI".Cage6_1.DB100_DBX137_1;
      AN    "Db Plc <=> HMI".Cage6_1.DB100_DBX137_2;
      AN    "Db Plc <=> HMI".Cage6_1.DB100_DBX137_6;
      AN    "Db Plc <=> HMI".Cage6_1.DB100_DBX137_7;
      AN    "Db Plc <=> HMI".Cage6_2.DB100_DBX138_0;
      AN    "Db Plc <=> HMI".Cage6_2.DB100_DBX138_1;
      AN    "Db Plc <=> HMI".Cage6_2.DB100_DBX138_2;
      AN    "Db Plc <=> HMI".Cage6_2.DB100_DBX138_3;
      AN    "Db Plc <=> HMI".Cage6_2.DB100_DBX138_4;
      AN    "Db Plc <=> HMI".Cage6_2.DB100_DBX138_5;
      AN    "Db Plc <=> HMI".Cage6_3.DB100_DBX141_6;
      AN    "Db Plc <=> HMI".Cage6_3.DB100_DBX141_7;
      AN    "Db Plc <=> HMI".Cage6_4.DB100_DBX142_0;
      AN    "Db Plc <=> HMI".Cage6_4.DB100_DBX142_1;
      AN    "Db Plc <=> HMI".Cage6_4.DB100_DBX142_2;
      AN    "Db Plc <=> HMI".Cage6_4.DB100_DBX142_3;
      AN    "Db Plc <=> HMI".Cage6_4.DB100_DBX142_4;
      AN    "Db Plc <=> HMI".Cage6_4.DB100_DBX142_5;
      AN    "Db Plc <=> HMI".Cage6_4.DB100_DBX142_6;
      AN    "Db Plc <=> HMI".Cage6_4.DB100_DBX142_7;
      AN    "Db Plc <=> HMI".Cage6_4.DB100_DBX143_0;
      ON    "M190.0";
      =     "M196.1";
END_FUNCTION

FUNCTION "Cage 6 unit" : VOID	// FC 30
TITLE = CAGE 6 UNIT FUNCTION
AUTHOR : Milesi
VERSION : 0.1
VAR_TEMP
  Brake_value : INT ;
END_VAR
BEGIN
NETWORK
TITLE = CAGE 6 OFF
      A(;
      L     "Cage 6".DB30_DBW2;
      L     0;
      ==I;
      );
      AN    "M180.1";
      AN    "M20.0";
      JNB   _001;
      R     "M190.0";
_001: NOP   0;
NETWORK
TITLE = CAGE 6 ON
      A(;
      L     "Cage 6".DB30_DBW2;
      L     1;
      ==I;
      );
      AN    "M180.1";
      AN    "M20.0";
      JNB   _040;
      S     "M190.0";
_040: NOP   0;
NETWORK
TITLE = CAGE 6 Z ROTATION
      A(;
      L     "Cage 6".DB30_DBW4;
      L     0;
      ==I;
      );
      AN    "M180.1";
      AN    "M20.0";
      JNB   _002;
      S     "M190.2";
      R     "M190.3";
_002: NOP   0;
NETWORK
TITLE = CAGE 6 S ROTATION
      A(;
      L     "Cage 6".DB30_DBW4;
      L     1;
      ==I;
      );
      AN    "M180.1";
      AN    "M20.0";
      JNB   _003;
      S     "M190.3";
      R     "M190.2";
_003: NOP   0;
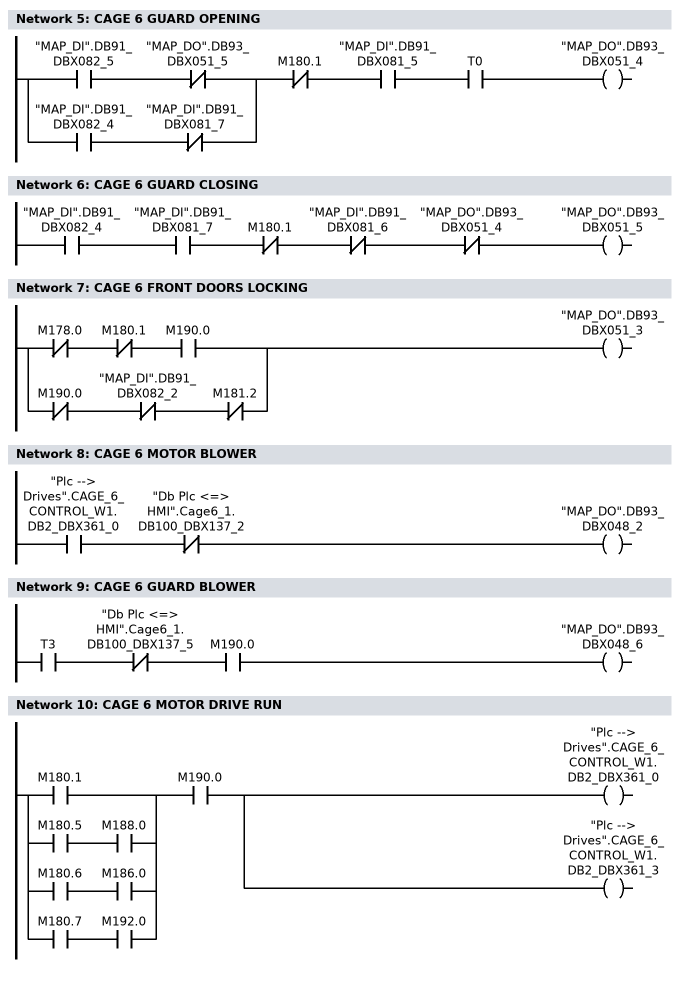
NETWORK
TITLE = CAGE 6 GUARD OPENING
      A(;
      A     "MAP_DI".DB91_DBX082_5;
      AN    "MAP_DO".DB93_DBX051_5;
      O;
      A     "MAP_DI".DB91_DBX082_4;
      AN    "MAP_DI".DB91_DBX081_7;
      );
      AN    "M180.1";
      A     "MAP_DI".DB91_DBX081_5;
      A     "T0";
      =     "MAP_DO".DB93_DBX051_4;
NETWORK
TITLE = CAGE 6 GUARD CLOSING
      A     "MAP_DI".DB91_DBX082_4;
      A     "MAP_DI".DB91_DBX081_7;
//      U     E     76.0
      AN    "M180.1";
      AN    "MAP_DI".DB91_DBX081_6;
      AN    "MAP_DO".DB93_DBX051_4;
      =     "MAP_DO".DB93_DBX051_5;
NETWORK
TITLE = CAGE 6 FRONT DOORS LOCKING
      AN    "M178.0";
      AN    "M180.1";
      A     "M190.0";
      O;
      AN    "M190.0";
      AN    "MAP_DI".DB91_DBX082_2;
      AN    "M181.2";
      =     "MAP_DO".DB93_DBX051_3;
NETWORK
TITLE = CAGE 6 MOTOR BLOWER 
      A     "Plc --> Drives".CAGE_6_CONTROL_W1.DB2_DBX361_0;
      AN    "Db Plc <=> HMI".Cage6_1.DB100_DBX137_2;
      =     "MAP_DO".DB93_DBX048_2;
NETWORK
TITLE = CAGE 6 GUARD BLOWER
      A     "T3";
      AN    "Db Plc <=> HMI".Cage6_1.DB100_DBX137_5;
      A     "M190.0";
      =     "MAP_DO".DB93_DBX048_6;
NETWORK
TITLE = CAGE 6 MOTOR DRIVE RUN
      A(;
      O     "M180.1";
      O;
      A     "M180.5";
      A     "M188.0";
      O;
      A     "M180.6";
      A     "M186.0";
      O;
      A     "M180.7";
      A     "M192.0";
      );
      A     "M190.0";
      =     "Plc --> Drives".CAGE_6_CONTROL_W1.DB2_DBX361_0;
      =     "Plc --> Drives".CAGE_6_CONTROL_W1.DB2_DBX361_3;
NETWORK
TITLE = CAGE 6 LAY SET ENABLE
      O     "M180.1";
      O     "M180.4";
      O(;
      A     "M180.5";
      A     "M188.0";
      );
      O(;
      A     "M180.6";
      A     "M186.0";
      );
      O(;
      A     "M180.7";
      A     "M192.0";
      );
      JC    _lay;
      L     "Cage 6".DB30_DBD20;
      T     "Cage 6".DB30_DBD24;
      JU    end1;
_lay: L     "Cage 6".DB30_DBD24;
      T     "Cage 6".DB30_DBD20;
end1: NOP   0;
NETWORK
TITLE = CAGE 6 MOTOR REFERENCE
//Max Linear Speed = 60 m/min
//Max Cage Rpm = 320
//
//Max Linear Speed              60000
//---------------- = Cage Lay = ----- = 187.5
//  Max Cage Rpm                 320
//
//                             Max Linear Speed
//Max Cage Rpm = 320 = 16384 = ---------------- * K
//                                Cage Lay
//
//    Cage Lay * 16384   187.5 * 16384
//K = ---------------- = ------------- = 51200
//    Max Linear Speed        60
// (network holds code this reader does not know; not shown)
NETWORK
TITLE = CAGE 6 MAX LINEAR SPEED TO START
      AN    "M200.1";
      JNB   _017;
      L     "Cage 6".DB30_DBD24;
      L     2.000000e-01;
      *R;
      JU    _018;
_017: L     "Cage 6".DB30_DBD24;
      L     2.600000e-01;
      *R;
_018: T     "Cage 6".DB30_DBD120;
      O(;
      L     6.000000e+01;
      >R;
      );
      ON    "M190.0";
      JNB   _014;
      T     "Cage 6".DB30_DBD120;
_014: NOP   0;
NETWORK
TITLE = CAGE 6 MAX LINEAR SPEED
      L     "Cage 6".DB30_DBD24;
      L     3.200000e-01;
      *R;
      T     "Cage 6".DB30_DBD96;
      O(;
      L     6.000000e+01;
      >R;
      );
      ON    "M190.0";
      JNB   _015;
      T     "Cage 6".DB30_DBD96;
_015: NOP   0;
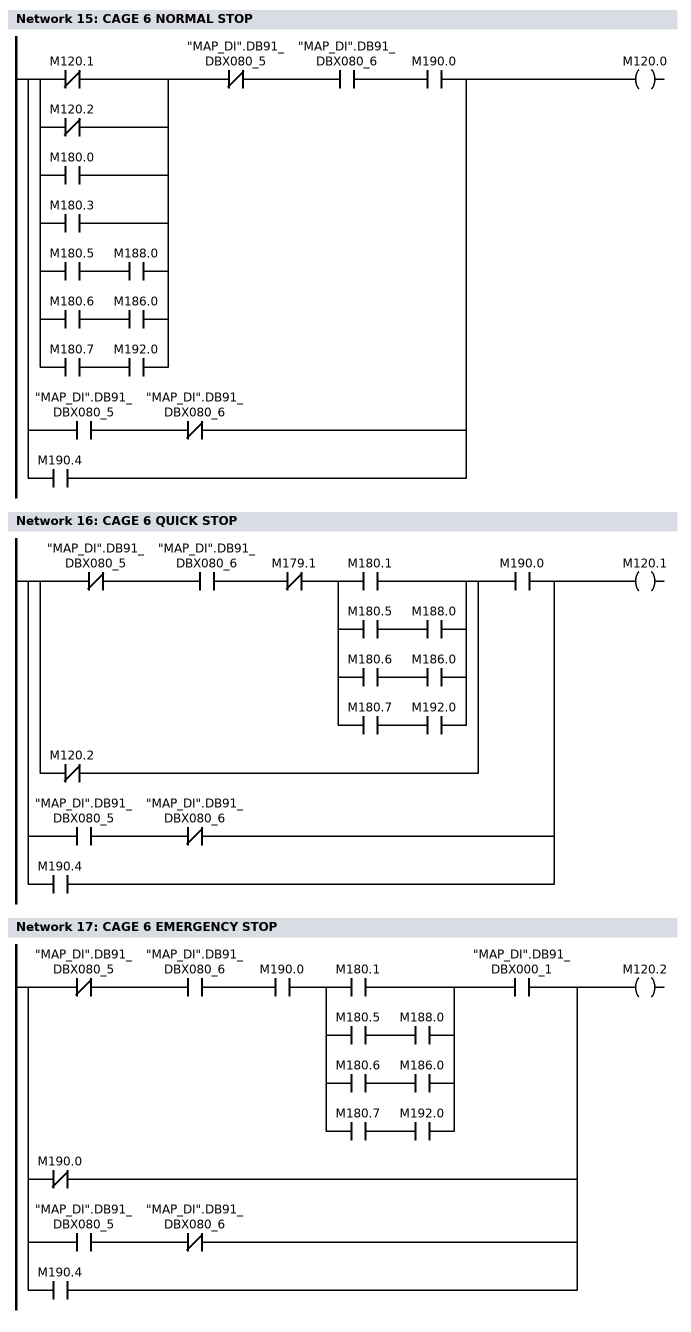
NETWORK
TITLE = CAGE 6 NORMAL STOP
      A(;
      ON    "M120.1";
      ON    "M120.2";
      O     "M180.0";
      O     "M180.3";
      O;
      A     "M180.5";
      A     "M188.0";
      O;
      A     "M180.6";
      A     "M186.0";
      O;
      A     "M180.7";
      A     "M192.0";
      );
      AN    "MAP_DI".DB91_DBX080_5;
      A     "MAP_DI".DB91_DBX080_6;
      A     "M190.0";
      O;
      A     "MAP_DI".DB91_DBX080_5;
      AN    "MAP_DI".DB91_DBX080_6;
      O     "M190.4";
      =     "M120.0";
NETWORK
TITLE = CAGE 6 QUICK STOP
      A(;
      AN    "MAP_DI".DB91_DBX080_5;
      A     "MAP_DI".DB91_DBX080_6;
      AN    "M179.1";
      A(;
      O     "M180.1";
      O;
      A     "M180.5";
      A     "M188.0";
      O;
      A     "M180.6";
      A     "M186.0";
      O;
      A     "M180.7";
      A     "M192.0";
      );
      ON    "M120.2";
      );
      A     "M190.0";
      O;
      A     "MAP_DI".DB91_DBX080_5;
      AN    "MAP_DI".DB91_DBX080_6;
      O     "M190.4";
      =     "M120.1";
NETWORK
TITLE = CAGE 6 EMERGENCY STOP
      AN    "MAP_DI".DB91_DBX080_5;
      A     "MAP_DI".DB91_DBX080_6;
      A     "M190.0";
      A(;
      O     "M180.1";
      O;
      A     "M180.5";
      A     "M188.0";
      O;
      A     "M180.6";
      A     "M186.0";
      O;
      A     "M180.7";
      A     "M192.0";
      );
      A     "MAP_DI".DB91_DBX000_1;
      ON    "M190.0";
      O;
      A     "MAP_DI".DB91_DBX080_5;
      AN    "MAP_DI".DB91_DBX080_6;
      O     "M190.4";
      =     "M120.2";
NETWORK
TITLE = CAGE 6 BRAKE PROPORTIONAL VALVE REFERENCE
      A     "M120.0";
      JC    _004;
      L     "Cage 6".DB30_DBD64;
      L     1.000000e+02;
      /R;
      L     2.764800e+04;
      *R;
      RND;
      JU    BRK;
_004: A     "M120.1";
      JC    _005;
      L     "Cage 6".DB30_DBD68;
      L     1.000000e+02;
      /R;
      L     2.764800e+04;
      *R;
      RND;
      JU    BRK;
_005: A     "M120.2";
      JC    _006;
      L     "Cage 6".DB30_DBD72;
      L     1.000000e+02;
      /R;
      L     2.764800e+04;
      *R;
      RND;
      JU    BRK;
_006: L     0;
BRK:  T     #Brake_value;
NETWORK
TITLE = SET POINT IN AMPER CALCULATION
      L     "Cage 6".DB20_DBD276;
      L     1.000000e+02;
      *R;
      L     1.000000e+02;
      /R;
      T     "Cage 6".DB20_DBD260;
NETWORK
TITLE = CURRENT CALCULATION
// (network holds code this reader does not know; not shown)
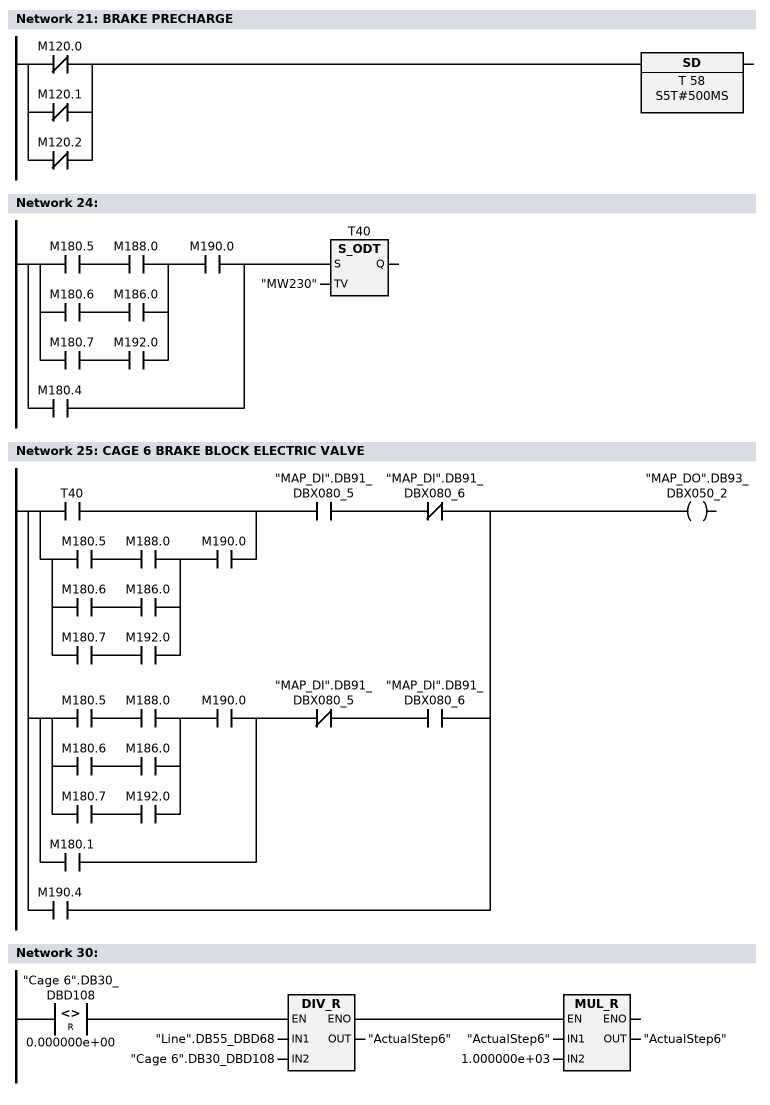
NETWORK
TITLE = BRAKE PRECHARGE
      ON    "M120.0";
      ON    "M120.1";
      ON    "M120.2";
      L     S5T#500MS;
      SD    T 58;
NETWORK
TITLE = BRAKE MODULATION CONTROL
      L     "Cage 6".DB20_DBD260;
      L     "Cage 6".DB30_DBD200;
      -R;
      T     "Cage 6".DB20_DBD264;
      L     "Cage 6".DB20_DBD268;
      *R;
      T     "Cage 6".DB20_DBD272;
      L     2.768400e+04;
      >R;
      JCN   _20d;
      L     2.768400e+04;
      T     "Cage 6".DB20_DBD272;
_20d: A     T 58;
      A     "M180.1";
      JCN   _20b;
      A(;
      L     "Cage 6".DB20_DBD272;
      L     0.000000e+00;
      <R;
      );
      JCN   _20a;
      L     0.000000e+00;
      T     "Cage 6".DB20_DBD272;
_20a: L     "Cage 6".DB20_DBD272;
      RND;
      JU    _20c;
_20b: L     #Brake_value;
_20c: T     "-359Y1";
NETWORK
TITLE = CAGE 6 BRAKE BLOCK OPEN ON-DELAY TIMER
      L     "Cage 6".DB30_DBD148;
      RND;
      ITB;
      L     W#16#2000;
      OW;
      T     "MW230";
NETWORK
TITLE =
      A(;
      A(;
      A     "M180.5";
      A     "M188.0";
      O;
      A     "M180.6";
      A     "M186.0";
      O;
      A     "M180.7";
      A     "M192.0";
      );
      A     "M190.0";
      O     "M180.4";
      );
      L     "MW230";
      SD    "T40";
      NOP   0;
      NOP   0;
      NOP   0;
      NOP   0;
NETWORK
TITLE = CAGE 6 BRAKE BLOCK ELECTRIC VALVE
      A(;
      O     "T40";
      O;
      A(;
      A     "M180.5";
      A     "M188.0";
      O;
      A     "M180.6";
      A     "M186.0";
      O;
      A     "M180.7";
      A     "M192.0";
      );
      A     "M190.0";
      );
      A     "MAP_DI".DB91_DBX080_5;
      AN    "MAP_DI".DB91_DBX080_6;
      O;
      A(;
      A(;
      A     "M180.5";
      A     "M188.0";
      O;
      A     "M180.6";
      A     "M186.0";
      O;
      A     "M180.7";
      A     "M192.0";
      );
      A     "M190.0";
      O     "M180.1";
      );
      AN    "MAP_DI".DB91_DBX080_5;
      A     "MAP_DI".DB91_DBX080_6;
      O     "M190.4";
      =     "MAP_DO".DB93_DBX050_2;
NETWORK
TITLE = CAGE 6 RPM TO HMI
      L     "Drives --> Plc".DB1_DBW366;
      ITD;
      DTR;
      L     1.638400e+04;
      /R;
      L     3.200000e+02;
      *R;
      ABS;
      T     "Cage 6".DB30_DBD108;
NETWORK
TITLE = CAGE 6 MOTOR RPM TO HMI
      L     "Drives --> Plc".DB1_DBW366;
      ITD;
      DTR;
      L     1.638400e+04;
      /R;
      L     1.495000e+03;
      *R;
      T     "Cage 6".DB30_DBD188;
NETWORK
TITLE = CAGE 6 MOTOR CURRENT TO HMI
      L     "Drives --> Plc".DB1_DBW368;
      ITD;
      DTR;
      L     1.638400e+04;
      /R;
      L     1.000000e+02;
      *R;
      T     "Cage 6".DB30_DBD192;
NETWORK
TITLE = CAGE 6 MOTOR VOLTAGE TO HMI
      L     "Drives --> Plc".DB1_DBW370;
      ITD;
      DTR;
      L     1.638400e+04;
      /R;
      L     4.000000e+02;
      *R;
      T     "Cage 6".DB30_DBD196;
NETWORK
TITLE =
      A(;
      A(;
      L     "Cage 6".DB30_DBD108;
      L     0.000000e+00;
      <>R;
      );
      JNB   _007;
      L     "Line".DB55_DBD68;
      L     "Cage 6".DB30_DBD108;
      /R;
      T     "ActualStep6";
      AN    OV;
      SAVE;
      CLR;
_007: A     BR;
      );
      JNB   _008;
      L     "ActualStep6";
      L     1.000000e+03;
      *R;
      T     "ActualStep6";
_008: NOP   0;
END_FUNCTION

FUNCTION "Cage 6 loading fase" : VOID	// FC 31
TITLE = CAGE 6 LOADING FASE FUNCTION
AUTHOR : Milesi
VERSION : 0.1
BEGIN
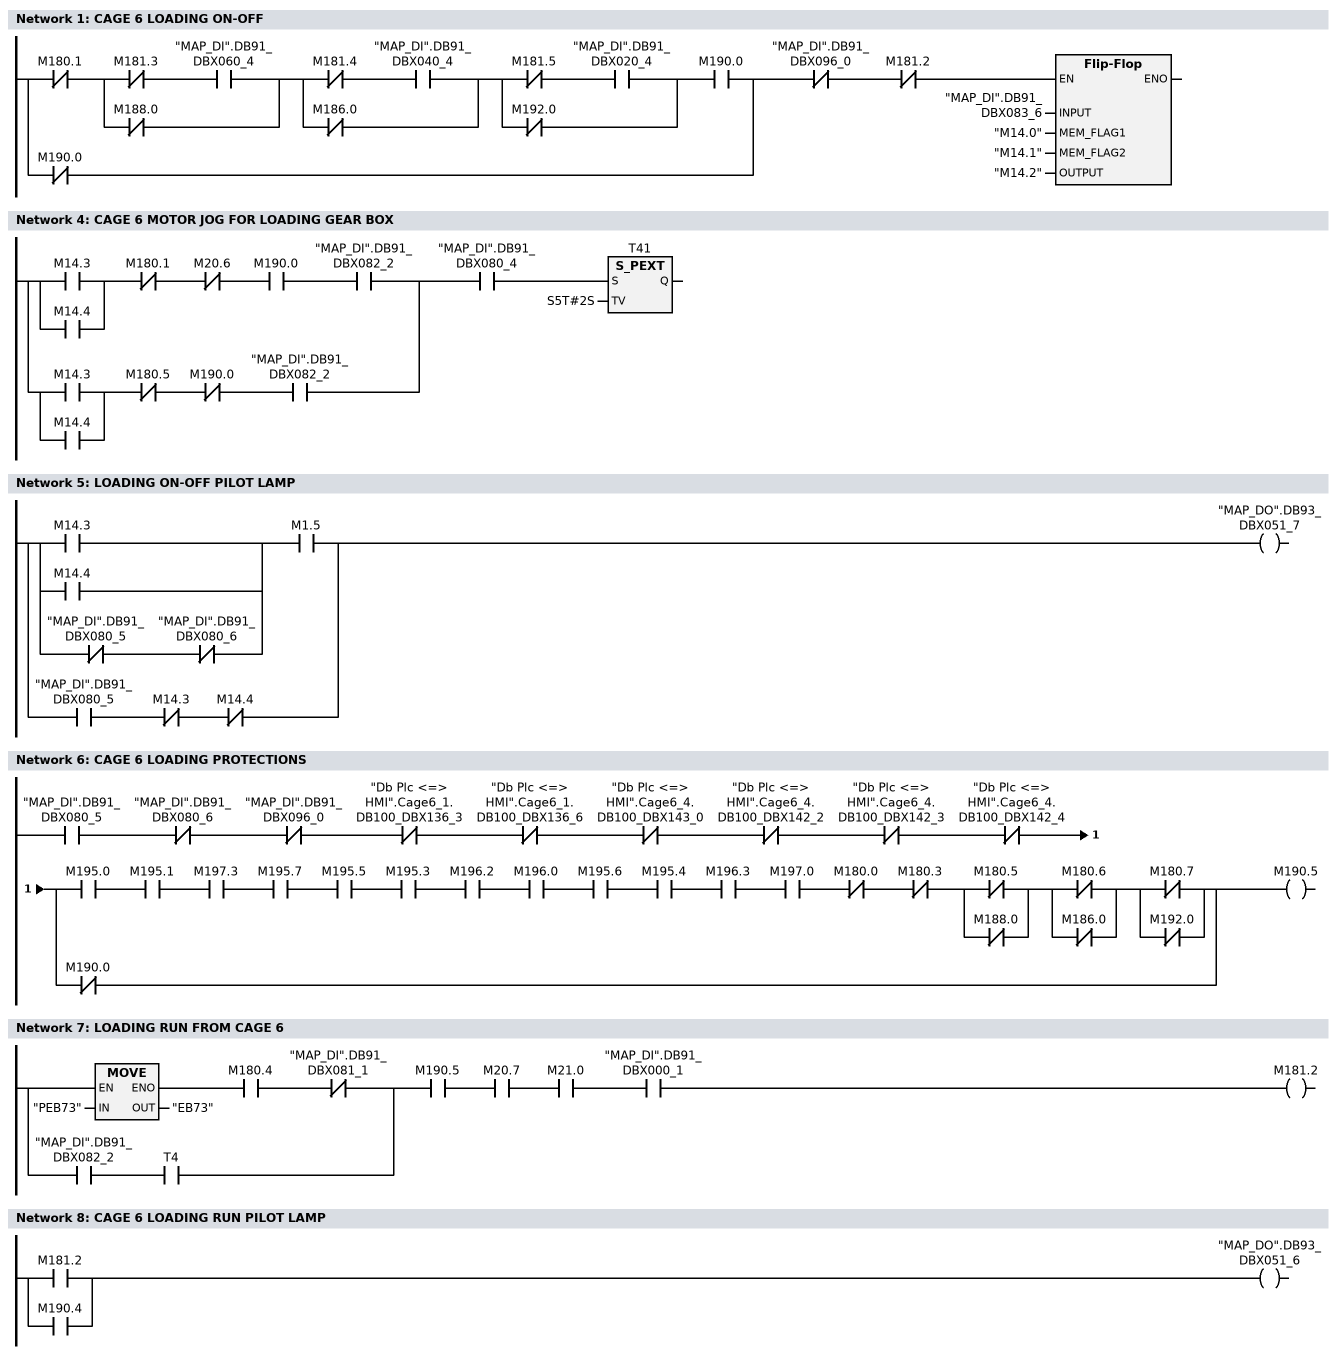
NETWORK
TITLE = CAGE 6 LOADING ON-OFF
      A(;
      AN    "M180.1";
      A(;
      AN    "M181.3";
      A     "MAP_DI".DB91_DBX060_4;
      ON    "M188.0";
      );
      A(;
      AN    "M181.4";
      A     "MAP_DI".DB91_DBX040_4;
      ON    "M186.0";
      );
      A(;
      AN    "M181.5";
      A     "MAP_DI".DB91_DBX020_4;
      ON    "M192.0";
      );
      A     "M190.0";
      ON    "M190.0";
      );
      AN    "MAP_DI".DB91_DBX096_0;
      AN    "M181.2";
      JNB   _001;
      CALL  "Flip-Flop" (
           INPUT                    := "MAP_DI".DB91_DBX083_6,
           MEM_FLAG1                := "M14.0",
           MEM_FLAG2                := "M14.1",
           OUTPUT                   := "M14.2");
_001: NOP   0;
NETWORK
TITLE = CAGE 6 LOADING ON
      A(;
      A(;
      A     "M14.2";
      AN    "M180.1";
      AN    "M20.6";
      A     "M190.0";
      O;
      AN    "M180.5";
      AN    "M190.0";
      );
      S     "MAP_DO".DB93_DBX050_0;
      A(;
      O     "MAP_DI".DB91_DBX080_5;
      O     "MAP_DO".DB93_DBX050_1;
      ON    "M14.2";
      );
      R     "MAP_DO".DB93_DBX050_0;
      A     "MAP_DO".DB93_DBX050_0;
      );
      S     "M14.3";
      A(;
      O     "MAP_DI".DB91_DBX080_5;
      ON    "M14.2";
      );
      R     "M14.3";
      NOP   0;
NETWORK
TITLE = CAGE 6 LOADING OFF
      A(;
      A(;
      AN    "M14.2";
      AN    "M20.6";
      A     "M190.0";
      O;
      AN    "M180.5";
      AN    "M190.0";
      );
      S     "MAP_DO".DB93_DBX050_1;
      A(;
      O     "MAP_DI".DB91_DBX080_6;
      O     "MAP_DO".DB93_DBX050_0;
      O     "M14.2";
      );
      R     "MAP_DO".DB93_DBX050_1;
      A     "MAP_DO".DB93_DBX050_1;
      );
      S     "M14.4";
      A(;
      O     "MAP_DI".DB91_DBX080_6;
      O     "M14.2";
      );
      R     "M14.4";
      NOP   0;
NETWORK
TITLE = CAGE 6 MOTOR JOG FOR LOADING GEAR BOX
      A(;
      A(;
      O     "M14.3";
      O     "M14.4";
      );
      AN    "M180.1";
      AN    "M20.6";
      A     "M190.0";
      A     "MAP_DI".DB91_DBX082_2;
      O;
      A(;
      O     "M14.3";
      O     "M14.4";
      );
      AN    "M180.5";
      AN    "M190.0";
      A     "MAP_DI".DB91_DBX082_2;
      );
      A     "MAP_DI".DB91_DBX080_4;
      L     S5T#2S;
      SE    "T41";
      NOP   0;
      NOP   0;
      NOP   0;
      NOP   0;
NETWORK
TITLE = LOADING ON-OFF PILOT LAMP
      A(;
      O     "M14.3";
      O     "M14.4";
      O;
      AN    "MAP_DI".DB91_DBX080_5;
      AN    "MAP_DI".DB91_DBX080_6;
      );
      A     "M1.5";
      O;
      A     "MAP_DI".DB91_DBX080_5;
      AN    "M14.3";
      AN    "M14.4";
      =     "MAP_DO".DB93_DBX051_7;
NETWORK
TITLE = CAGE 6 LOADING PROTECTIONS
      A     "MAP_DI".DB91_DBX080_5;
      AN    "MAP_DI".DB91_DBX080_6;
      AN    "MAP_DI".DB91_DBX096_0;
      AN    "Db Plc <=> HMI".Cage6_1.DB100_DBX136_3;
      AN    "Db Plc <=> HMI".Cage6_1.DB100_DBX136_6;
      AN    "Db Plc <=> HMI".Cage6_4.DB100_DBX143_0;
      AN    "Db Plc <=> HMI".Cage6_4.DB100_DBX142_2;
      AN    "Db Plc <=> HMI".Cage6_4.DB100_DBX142_3;
      AN    "Db Plc <=> HMI".Cage6_4.DB100_DBX142_4;
      A(;
      A     "M195.0";
      A     "M195.1";
      A     "M197.3";
      A     "M195.7";
      A     "M195.5";
      A     "M195.3";
      A     "M196.2";
      A     "M196.0";
      A     "M195.6";
      A     "M195.4";
      A     "M196.3";
      A     "M197.0";
      AN    "M180.0";
      AN    "M180.3";
      A(;
      ON    "M180.5";
      ON    "M188.0";
      );
      A(;
      ON    "M180.6";
      ON    "M186.0";
      );
      A(;
      ON    "M180.7";
      ON    "M192.0";
      );
      ON    "M190.0";
      );
      =     "M190.5";
NETWORK
TITLE = LOADING RUN FROM CAGE 6
      A(;
      A(;
      L     "PEB73";
      T     "EB73";
      SET;
      SAVE;
      CLR;
      A     BR;
      );
      A     "M180.4";
      AN    "MAP_DI".DB91_DBX081_1;
      O;
      A     "MAP_DI".DB91_DBX082_2;
      A     "T4";
      );
      A     "M190.5";
      A     "M20.7";
      A     "M21.0";
      A     "MAP_DI".DB91_DBX000_1;
      =     "M181.2";
NETWORK
TITLE = CAGE 6 LOADING RUN PILOT LAMP
      O     "M181.2";
      O     "M190.4";
      =     "MAP_DO".DB93_DBX051_6;
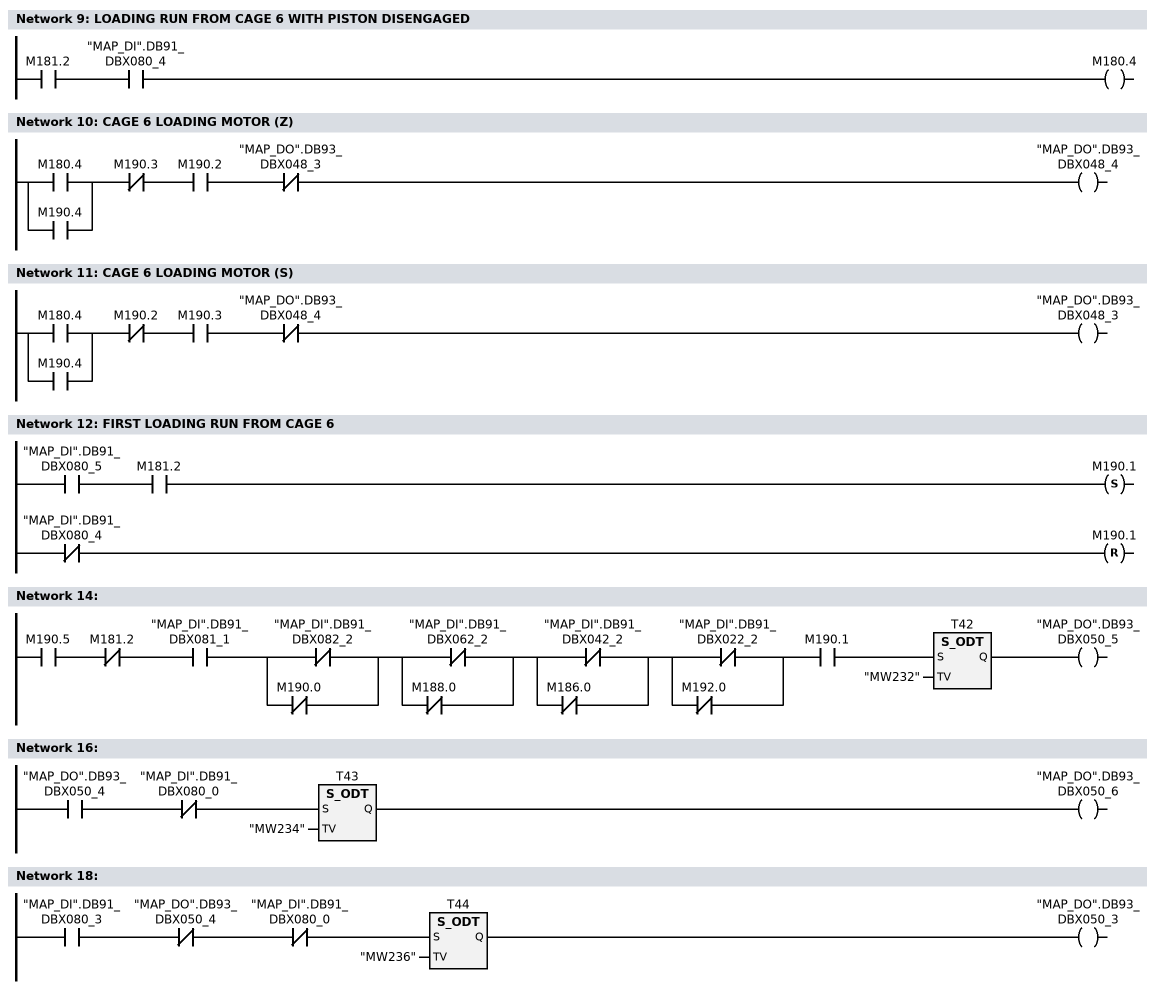
NETWORK
TITLE = LOADING RUN FROM CAGE 6 WITH PISTON DISENGAGED
      A     "M181.2";
      A     "MAP_DI".DB91_DBX080_4;
      =     "M180.4";
NETWORK
TITLE = CAGE 6 LOADING MOTOR (Z)
      A(;
      O     "M180.4";
      O     "M190.4";
      );
      AN    "M190.3";
      A     "M190.2";
      AN    "MAP_DO".DB93_DBX048_3;
      =     "MAP_DO".DB93_DBX048_4;
NETWORK
TITLE = CAGE 6 LOADING MOTOR (S)
      A(;
      O     "M180.4";
      O     "M190.4";
      );
      AN    "M190.2";
      A     "M190.3";
      AN    "MAP_DO".DB93_DBX048_4;
      =     "MAP_DO".DB93_DBX048_3;
NETWORK
TITLE = FIRST LOADING RUN FROM CAGE 6
      A     "MAP_DI".DB91_DBX080_5;
      A     "M181.2";
      S     "M190.1";
      AN    "MAP_DI".DB91_DBX080_4;
      R     "M190.1";
      NOP   0;
NETWORK
TITLE = CAGE 6 PISTON ENGAGING INTO CAGE
      L     "Cage 6".DB30_DBD152;
      RND;
      ITB;
      L     W#16#2000;
      OW;
      T     "MW232";
NETWORK
TITLE =
      A     "M190.5";
      AN    "M181.2";
      A     "MAP_DI".DB91_DBX081_1;
      A(;
      ON    "MAP_DI".DB91_DBX082_2;
      ON    "M190.0";
      );
      A(;
      ON    "MAP_DI".DB91_DBX062_2;
      ON    "M188.0";
      );
      A(;
      ON    "MAP_DI".DB91_DBX042_2;
      ON    "M186.0";
      );
      A(;
      ON    "MAP_DI".DB91_DBX022_2;
      ON    "M192.0";
      );
      A     "M190.1";
      L     "MW232";
      SD    "T42";
      NOP   0;
      NOP   0;
      NOP   0;
      A     "T42";
      =     "MAP_DO".DB93_DBX050_5;
NETWORK
TITLE = CAGE 6 PISTON DISENGAGING FROM CAGE
      L     "Cage 6".DB30_DBD144;
      RND;
      ITB;
      L     W#16#2000;
      OW;
      T     "MW234";
NETWORK
TITLE =
      A     "MAP_DO".DB93_DBX050_4;
      AN    "MAP_DI".DB91_DBX080_0;
      L     "MW234";
      SD    "T43";
      NOP   0;
      NOP   0;
      NOP   0;
      A     "T43";
      =     "MAP_DO".DB93_DBX050_6;
NETWORK
TITLE = CAGE 6 AIR INLET INTO CAGE
      L     "Cage 6".DB30_DBD156;
      RND;
      ITB;
      L     W#16#2000;
      OW;
      T     "MW236";
NETWORK
TITLE =
      A     "MAP_DI".DB91_DBX080_3;
      AN    "MAP_DO".DB93_DBX050_4;
      AN    "MAP_DI".DB91_DBX080_0;
      L     "MW236";
      SD    "T44";
      NOP   0;
      NOP   0;
      NOP   0;
      A     "T44";
      =     "MAP_DO".DB93_DBX050_3;
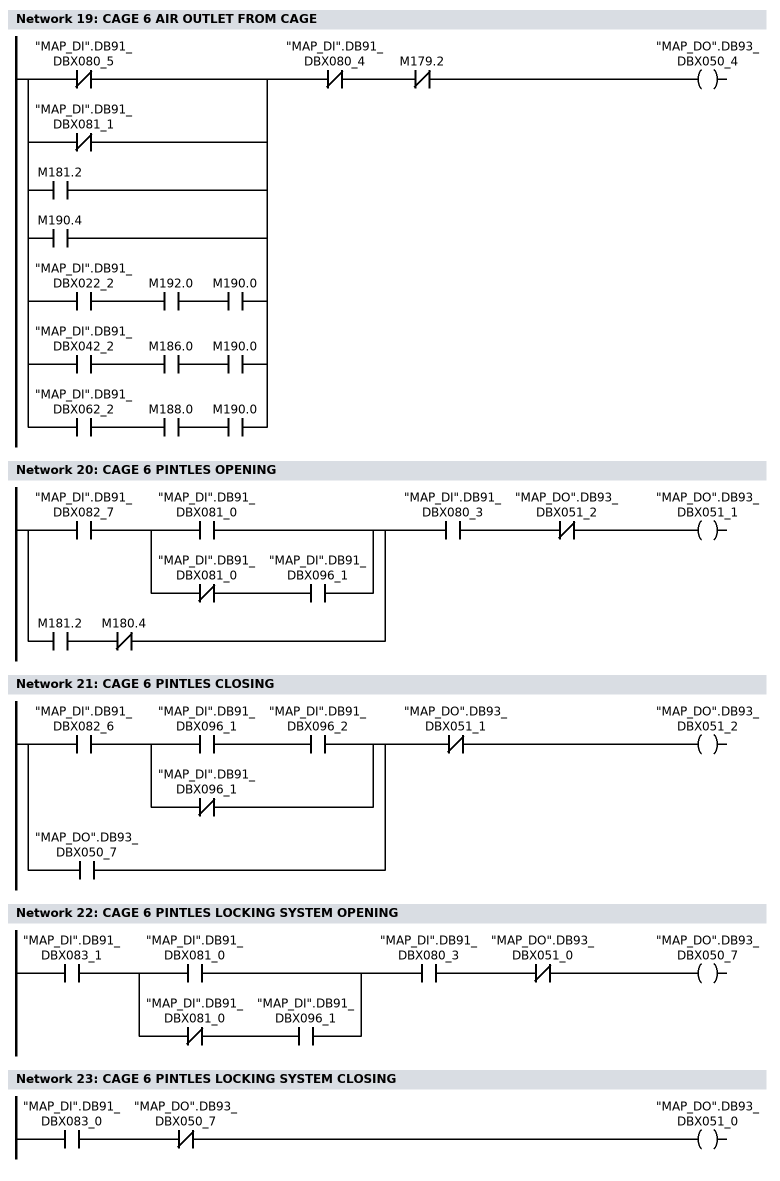
NETWORK
TITLE = CAGE 6 AIR OUTLET FROM CAGE
      A(;
      ON    "MAP_DI".DB91_DBX080_5;
      ON    "MAP_DI".DB91_DBX081_1;
      O     "M181.2";
      O     "M190.4";
      O;
      A     "MAP_DI".DB91_DBX022_2;
      A     "M192.0";
      A     "M190.0";
      O;
      A     "MAP_DI".DB91_DBX042_2;
      A     "M186.0";
      A     "M190.0";
      O;
      A     "MAP_DI".DB91_DBX062_2;
      A     "M188.0";
      A     "M190.0";
      );
      AN    "MAP_DI".DB91_DBX080_4;
      AN    "M179.2";
      =     "MAP_DO".DB93_DBX050_4;
NETWORK
TITLE = CAGE 6 PINTLES OPENING
      A(;
      A     "MAP_DI".DB91_DBX082_7;
      A(;
      O     "MAP_DI".DB91_DBX081_0;
      O;
      AN    "MAP_DI".DB91_DBX081_0;
      A     "MAP_DI".DB91_DBX096_1;
      );
      O;
      A     "M181.2";
      AN    "M180.4";
      );
      A     "MAP_DI".DB91_DBX080_3;
      AN    "MAP_DO".DB93_DBX051_2;
      =     "MAP_DO".DB93_DBX051_1;
NETWORK
TITLE = CAGE 6 PINTLES CLOSING
      A(;
      A     "MAP_DI".DB91_DBX082_6;
      A(;
      A     "MAP_DI".DB91_DBX096_1;
      A     "MAP_DI".DB91_DBX096_2;
      ON    "MAP_DI".DB91_DBX096_1;
      );
      O     "MAP_DO".DB93_DBX050_7;
      );
      AN    "MAP_DO".DB93_DBX051_1;
      =     "MAP_DO".DB93_DBX051_2;
NETWORK
TITLE = CAGE 6 PINTLES LOCKING SYSTEM OPENING
      A     "MAP_DI".DB91_DBX083_1;
      A(;
      O     "MAP_DI".DB91_DBX081_0;
      O;
      AN    "MAP_DI".DB91_DBX081_0;
      A     "MAP_DI".DB91_DBX096_1;
      );
      A     "MAP_DI".DB91_DBX080_3;
      AN    "MAP_DO".DB93_DBX051_0;
      =     "MAP_DO".DB93_DBX050_7;
NETWORK
TITLE = CAGE 6 PINTLES LOCKING SYSTEM CLOSING
      A     "MAP_DI".DB91_DBX083_0;
      AN    "MAP_DO".DB93_DBX050_7;
      =     "MAP_DO".DB93_DBX051_0;
NETWORK
TITLE = CAGE 6 PLATFORM UP
NETWORK
TITLE = CAGE 6 PLATFORM DOWN
NETWORK
TITLE = CAGE 6 EVEN BOBBINS ROTATION FOR LOADING MACHINE
NETWORK
TITLE = CAGE 6 EVEN BOBBINS ROTATION FOR LOADING PLATFORM
NETWORK
TITLE = CAGE 6 ODD BOBBINS ROTATION FOR LOADING MACHINE
NETWORK
TITLE = CAGE 6 ODD BOBBINS ROTATION FOR LOADING PLATFORM
NETWORK
TITLE = CAGE 6 BOBBIN ROTATION FOR LOADING MACHINE PILOT LAMP
NETWORK
TITLE = CAGE 6 LOADING PUMP
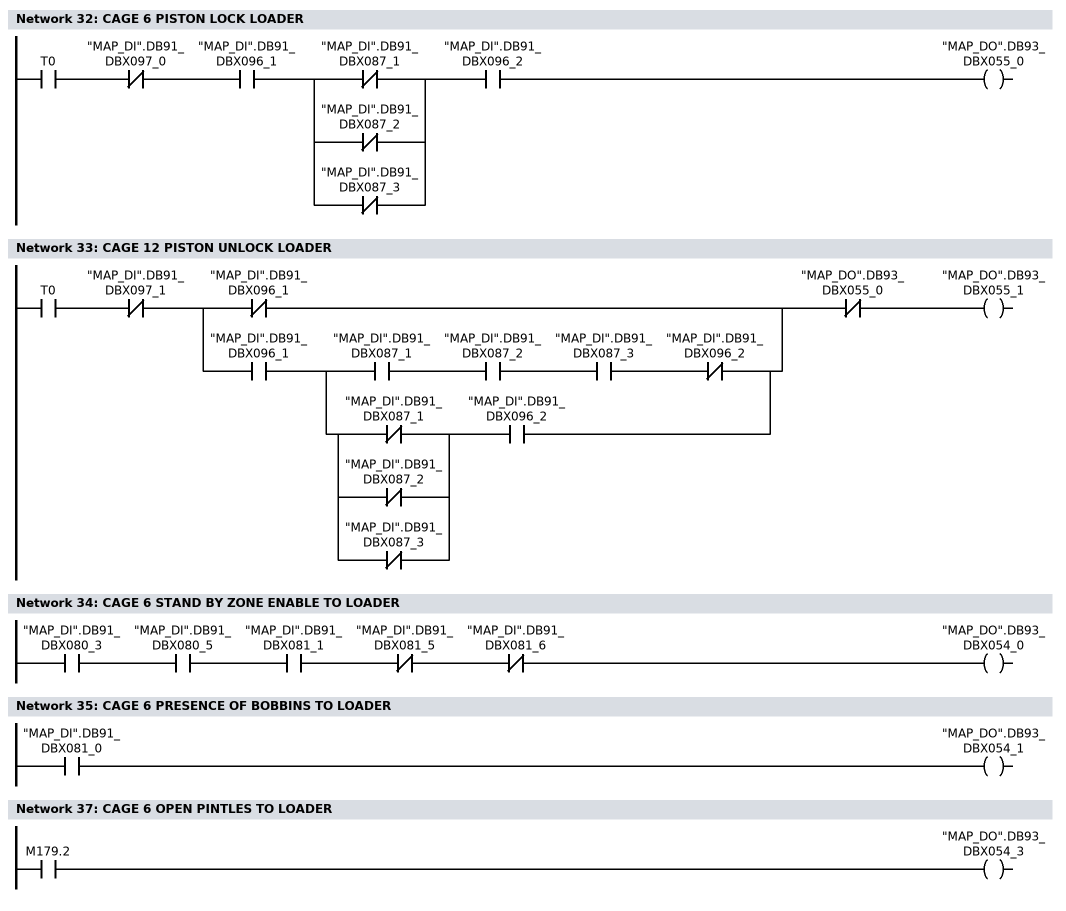
NETWORK
TITLE = CAGE 6 PISTON LOCK LOADER
      A     "T0";
      AN    "MAP_DI".DB91_DBX097_0;
      A     "MAP_DI".DB91_DBX096_1;
      A(;
      ON    "MAP_DI".DB91_DBX087_1;
      ON    "MAP_DI".DB91_DBX087_2;
      ON    "MAP_DI".DB91_DBX087_3;
      );
      A     "MAP_DI".DB91_DBX096_2;
      =     "MAP_DO".DB93_DBX055_0;
NETWORK
TITLE = CAGE 12 PISTON UNLOCK LOADER
      A     "T0";
      AN    "MAP_DI".DB91_DBX097_1;
      A(;
      ON    "MAP_DI".DB91_DBX096_1;
      O;
      A     "MAP_DI".DB91_DBX096_1;
      A(;
      A     "MAP_DI".DB91_DBX087_1;
      A     "MAP_DI".DB91_DBX087_2;
      A     "MAP_DI".DB91_DBX087_3;
      AN    "MAP_DI".DB91_DBX096_2;
      O;
      A(;
      ON    "MAP_DI".DB91_DBX087_1;
      ON    "MAP_DI".DB91_DBX087_2;
      ON    "MAP_DI".DB91_DBX087_3;
      );
      A     "MAP_DI".DB91_DBX096_2;
      );
      );
      AN    "MAP_DO".DB93_DBX055_0;
      =     "MAP_DO".DB93_DBX055_1;
NETWORK
TITLE = CAGE 6 STAND BY ZONE ENABLE TO LOADER
      A     "MAP_DI".DB91_DBX080_3;
      A     "MAP_DI".DB91_DBX080_5;
      A     "MAP_DI".DB91_DBX081_1;
      AN    "MAP_DI".DB91_DBX081_5;
      AN    "MAP_DI".DB91_DBX081_6;
      =     "MAP_DO".DB93_DBX054_0;
NETWORK
TITLE = CAGE 6 PRESENCE OF BOBBINS TO LOADER
      A     "MAP_DI".DB91_DBX081_0;
      =     "MAP_DO".DB93_DBX054_1;
NETWORK
TITLE = CAGE 6 LOADER LOCK PISTON INSERTED TO LOADER 
      CLR;
      =     "MAP_DO".DB93_DBX054_2;
NETWORK
TITLE = CAGE 6 OPEN PINTLES TO LOADER
      A     "M179.2";
      =     "MAP_DO".DB93_DBX054_3;
END_FUNCTION

FUNCTION "Cage 6 preforming alarms" : VOID	// FC 32
TITLE = CAGE 6 PREFORMING ALARMS FUNCTION
AUTHOR : Milesi
VERSION : 0.1
BEGIN
NETWORK
TITLE = CAGE 12 PREFORMING OPEN GUARD - NOT USED
//NOT USED
      A     "T0";
      A     "M180.1";
      AN    "MAP_DI".DB91_DBX084_6;
      CLR;
      S     "M174.6";
NETWORK
TITLE =
//NOT USED
      A     "T0";
      A(;
      ON    "MAP_DI".DB91_DBX084_6;
      O     "M174.6";
      );
      CLR;
      =     "Db Plc <=> HMI".Cage6_4.DB100_DBX143_6;
NETWORK
TITLE = CAGE 6 PREFORMING GENERAL ALARM
      AN    "Db Plc <=> HMI".Cage6_4.DB100_DBX143_6;
      =     "M196.2";
END_FUNCTION

FUNCTION "Cage 6 preforming unit" : VOID	// FC 33
TITLE = CAGE 6 PREFORMING UNIT FUNCTION
AUTHOR : Milesi
VERSION : 0.1
BEGIN
// (block stored without names or comments; labels and parameter names are numbered)
END_FUNCTION

FUNCTION "Pay-off 630 alarms" : VOID	// FC 34
TITLE = PAY-OFF 630 ALARMS FUNCTION
AUTHOR : Milesi
VERSION : 0.1
VAR_TEMP
  EnableWireBreakAlarm : BOOL ;
  aux1 : BOOL ;
  aux2 : BOOL ;
  aux3 : INT ;
END_VAR
BEGIN
NETWORK
TITLE = PAY-OFF 630 OPEN PINTLES ALARM
      A     "T0";
      A     "M180.1";
      AN    "MAP_DI".DB91_DBX099_0;
      A     "Pay-off 630".HMI_Bit.DB35_DBX1_7;
      S     "M175.2";
NETWORK
TITLE =
      A     "T0";
      A(;
      ON    "MAP_DI".DB91_DBX099_0;
      O     "M175.2";
      );
      A     "Pay-off 630".HMI_Bit.DB35_DBX1_7;
      =     "Db Plc <=> HMI".CENTRAL_PAY_OFF.DB100_DBX147_00;
NETWORK
TITLE = PAY-OFF 630 BOBBIN WIRE BREAK
      A     "M201.2";
      A     "Pay-off 630".HMI_Bit.DB35_DBX1_1;
      A     "Pay-off 630".HMI_Bit.DB35_DBX1_7;
      =     #EnableWireBreakAlarm;
      CALL  "Rotation control" (
           Enable                   := #EnableWireBreakAlarm,
           Pulse                    := "MAP_DI".DB91_DBX099_1,
           Reset                    := "M30.1",
           DelayTime                := "Pay-off 630".DB35_DBW6,
           StorageTimer             := "T160",
           Mem                      := "M175.3",
           ALARM                    := "Db Plc <=> HMI".CENTRAL_PAY_OFF.DB100_DBX147_01);
      A     "Db Plc <=> HMI".CENTRAL_PAY_OFF.DB100_DBX147_01;
      =     "MAP_DO".DB93_DBX058_0;
NETWORK
TITLE = PAY-OFF 630 MAIN AIR MINIMUM PRESSURE
      A     "T0";
      A     "M180.1";
      AN    "MAP_DI".DB91_DBX099_2;
      A     "Pay-off 630".HMI_Bit.DB35_DBX1_7;
      S     "M175.4";
NETWORK
TITLE =
      A     "T0";
      A(;
      ON    "MAP_DI".DB91_DBX099_2;
      O     "M175.4";
      );
      A     "Pay-off 630".HMI_Bit.DB35_DBX1_7;
      =     "Db Plc <=> HMI".CENTRAL_PAY_OFF.DB100_DBX147_02;
NETWORK
TITLE = PAY-OFF 630 BRAKE OFF
      A     "T0";
      A     "M180.1";
      A     "MAP_DI".DB91_DBX099_4;
      A     "Pay-off 630".HMI_Bit.DB35_DBX1_7;
      S     "M175.5";
NETWORK
TITLE =
      A     "T0";
      A(;
      O     "MAP_DI".DB91_DBX099_4;
      O     "M175.5";
      );
      A     "Pay-off 630".HMI_Bit.DB35_DBX1_7;
      =     "Db Plc <=> HMI".CENTRAL_PAY_OFF.DB100_DBX147_03;
NETWORK
TITLE = PAY-OFF 630 GENERAL ALARM
      AN    "Db Plc <=> HMI".CENTRAL_PAY_OFF.DB100_DBX147_00;
      AN    "Db Plc <=> HMI".CENTRAL_PAY_OFF.DB100_DBX147_01;
      AN    "Db Plc <=> HMI".CENTRAL_PAY_OFF.DB100_DBX147_02;
      AN    "Db Plc <=> HMI".CENTRAL_PAY_OFF.DB100_DBX147_03;
      =     "M196.3";
END_FUNCTION

FUNCTION "Pay-off 630 unit" : VOID	// FC 35
TITLE = PAY-OFF 630 UNIT FUNCTION
AUTHOR : Milesi
VERSION : 0.1
BEGIN
NETWORK
TITLE = PAY-OFF 630 INSERTION
      A     "Pay-off 630".HMI_Bit.DB35_DBX1_0;
      AN    "M180.1";
      AN    "M20.6";
      S     "Pay-off 630".HMI_Bit.DB35_DBX1_7;
      AN    "Pay-off 630".HMI_Bit.DB35_DBX1_0;
      AN    "M180.1";
      AN    "M20.6";
      R     "Pay-off 630".HMI_Bit.DB35_DBX1_7;
NETWORK
TITLE = PAY-OFF 630 PINTLES ENABLE
      AN    "M180.1";
      =     "MAP_DO".DB93_DBX058_2;
NETWORK
TITLE = PAY-OFF 630 PINTLES OPEN PILOT LAMP
      AN    "MAP_DI".DB91_DBX099_0;
      =     "MAP_DO".DB93_DBX058_1;
END_FUNCTION

FUNCTION "Metercounter alarms" : VOID	// FC 40
TITLE = METERCOUNTER ALARMS FUNCTION
AUTHOR : Milesi
VERSION : 0.1
VAR_TEMP
  Impulses_encoder : DINT ;
  Metercounter_K : REAL ;
END_VAR
BEGIN
NETWORK
TITLE = LINE SLOW-DOWN FROM METERCOUNTER
      A     "T0";
      A(;
      L     "Metercounter".DB41_DBD52;
      L     "Metercounter".DB41_DBD36;
      <=R;
      );
      AN    "Db Plc <=> HMI".LINE1.DB100_DBX148_0;
      =     "Db Plc <=> HMI".LINE1.DB100_DBX149_7;
NETWORK
TITLE = LINE STOP FROM METERCOUNTER
      A     "T0";
      A(;
      L     "Metercounter".DB41_DBD44;
      L     "Metercounter".DB41_DBD32;
      >=R;
      );
      S     "Db Plc <=> HMI".LINE1.DB100_DBX148_0;
NETWORK
TITLE = METERCOUNTER GENERAL ALARM
      AN    "Db Plc <=> HMI".LINE1.DB100_DBX148_0;
      =     "M196.7";
END_FUNCTION

FUNCTION "Metercounter unit" : VOID	// FC 41
TITLE = METERCOUNTER UNIT FUNCTION
AUTHOR : Milesi
VERSION : 0.1
VAR_TEMP
  Metercounter_encoder_imp : DINT ;
  Constant_m_for_imp : REAL ;
  Encoder_imp : REAL ;
END_VAR
BEGIN
NETWORK
TITLE = METERCOUNTER ENCODER COUNTER
      L     "PED260";
      NEGD;
      T     #Metercounter_encoder_imp;
NETWORK
TITLE = METERCOUNTER CALCULATION (m/imp)
//capstan pulley Ш + cable Ш * 3.1415              mm/imp
//------------------------------------ = mm/imp = -------- = m/imp
//capstan gear ratio * encoder imp * 4              1000
//
      L     2.406828e+02;
      L     1.024000e+03;
      *R;
      L     4.000000e+00;
      *R;
      T     #Encoder_imp;
      L     2.500000e+03;
      L     "Line".DB55_DBD56;
      +R;
      L     3.141593e+00;
      *R;
      L     #Encoder_imp;
      /R;
      L     1.000000e+03;
      /R;
      T     #Constant_m_for_imp;
NETWORK
TITLE = METERCOUNTER METERS INCREASE
      L     #Metercounter_encoder_imp;
      L     "Metercounter".DB41_DBD132;
      -D;
      DTR;
      L     #Constant_m_for_imp;
      *R;
      L     "Metercounter".DB41_DBD48;
      *R;
      T     "Metercounter".DB41_DBD72;
      L     #Metercounter_encoder_imp;
      T     "Metercounter".DB41_DBD132;
NETWORK
TITLE = ACTUAL LENGHT
      A     "M180.1";
      JCN   _gi1;
      L     "Metercounter".DB41_DBD72;
      L     "Metercounter".DB41_DBD44;
      +R;
      T     "Metercounter".DB41_DBD44;
_gi1: NOP   0;
NETWORK
TITLE = ACTUAL TOTAL LENGHT
      A     "M180.1";
      JCN   _gi2;
      L     "Metercounter".DB41_DBD72;
      L     "Metercounter".DB41_DBD40;
      +R;
      T     "Metercounter".DB41_DBD40;
_gi2: NOP   0;
NETWORK
TITLE = LENGTH TO MAKE
      L     "Metercounter".DB41_DBD32;
      L     "Metercounter".DB41_DBD44;
      -R;
      T     "Metercounter".DB41_DBD52;
      NOP   0;
NETWORK
TITLE = ACTUAL LENGHT RESET
      A     "Metercounter".HMI_Bit.DB41_DBX1_0;
      JNB   _004;
      L     0.000000e+00;
      T     "Metercounter".DB41_DBD44;
      T     "Metercounter".DB41_DBD111;
_004: NOP   0;
NETWORK
TITLE = ACTUAL TOTAL LENGHT RESET
      A     "Metercounter".HMI_Bit.DB41_DBX1_1;
      JNB   _005;
      L     0.000000e+00;
      T     "Metercounter".DB41_DBD40;
_005: NOP   0;
NETWORK
TITLE =
      A     "M3.0";
      JCN   m09a;
      L     "Capstan".DB9_DBD188;
      L     6.000000e+01;
      /R;
      L     1.000000e-01;
      *R;
      T     "Metercounter".DB41_DBD100;
      L     2.500000e+03;
      L     "Line".DB55_DBD56;
      +R;
      T     "Metercounter".DB41_DBD104;
      L     1.000000e+03;
      /R;
      L     "Metercounter".DB41_DBD100;
      *R;
      L     3.141593e+00;
      *R;
      L     2.406828e+02;
      /R;
      T     "Metercounter".DB41_DBD108;
      L     "Metercounter".DB41_DBD108;
      L     "Metercounter".DB41_DBD111;
      +R;
      T     "Metercounter".DB41_DBD111;
      L     "Metercounter".DB41_DBD111;
      L     "Metercounter".DB41_DBD44;
      -R;
      T     "Metercounter".DB41_DBD116;
m09a: NOP   0;
NETWORK
TITLE = TEST CAPSTAN DIRECT LENGHT MAKE
      L     "Capstan".DB9_DBD188;
END_FUNCTION

FUNCTION "Common function" : VOID	// FC 50
TITLE = COMMON FUNCTION UNIT
AUTHOR : Milesi
VERSION : 0.1
VAR_TEMP
  T2_time : S5TIME ;	//T2 BCD time set from MP
  T1_time : S5TIME ;	//T5 BCD time set from MP
END_VAR
BEGIN
NETWORK
TITLE =  IMPULSO 100 MILLISECONDI
      A     "M1.0";
      FP    "M2.0";
      =     "M3.0";
NETWORK
TITLE =  IMPULSO 200 MILLISECONDI
      A     "M1.1";
      FP    "M2.1";
      =     "M3.1";
NETWORK
TITLE =  IMPULSO 400 MILLISECONDI
      A     "M1.2";
      FP    "M2.2";
      =     "M3.2";
NETWORK
TITLE =  IMPULSO 500 MILLISECONDI
      A     "M1.3";
      FP    "M2.3";
      =     "M3.3";
NETWORK
TITLE =  IMPULSO 800 MILLISECONDI
      A     "M1.4";
      FP    "M2.4";
      =     "M3.4";
NETWORK
TITLE =  IMPULSO  1 SECONDO
      A     "M1.5";
      FP    "M2.5";
      =     "M3.5";
NETWORK
TITLE =  IMPULSO 1,6 SECONDI
      A     "M1.6";
      FP    "M2.6";
      =     "M3.6";
NETWORK
TITLE = IMPULSO  2 SECONDI
      A     "M1.7";
      FP    "M2.7";
      =     "M3.7";
NETWORK
TITLE = PLC<-->OP COMUNICATION ON CONTROL
      AN    "M1.6";
      =     "M30.0";
NETWORK
TITLE = SYNCHRONIZATION PLC<-->OP FOR DATA TRANSFER
      A     "M180.1";
      JC    LAB1;
      A     DB100.DBX 7.2;
      R     DB100.DBX 7.2;
      JU    LAB2;
LAB1: =     DB100.DBX 7.2;
LAB2: NOP   0;
END_FUNCTION

FUNCTION "Hour counter" : VOID	// FC 51
TITLE = HOURS COUNTER FUNCTION
AUTHOR : Milesi
VERSION : 0.1
BEGIN
NETWORK
TITLE = HOUR COUNTER SECOND INCREASE
      ON    "M180.0";
      ON    "M3.5";
      JC    _001;
      L     "Line".DB55_DBD20;
      L     1.000000e+00;
      +R;
      T     "Line".DB55_DBD20;
_001: NOP   0;
NETWORK
TITLE = HOUR COUNTER HOUR INCREASE
      A(;
      L     "Line".DB55_DBD20;
      L     3.600000e+03;
      <=R;
      );
      JC    _002;
      L     "Line".DB55_DBD24;
      L     1.000000e+00;
      +R;
      T     "Line".DB55_DBD24;
      L     0.000000e+00;
      T     "Line".DB55_DBD20;
_002: NOP   0;
END_FUNCTION

FUNCTION "Line alarms" : VOID	// FC 52
TITLE = LINE ALARMS FUNCTION
AUTHOR : Milesi
VERSION : 0.1
BEGIN
NETWORK
TITLE = AUXILIARY OFF ALARM
      AN    "MAP_DI".DB91_DBX000_0;
      =     "Db Plc <=> HMI".LINE1.DB100_DBX149_0;
NETWORK
TITLE = EMERGENCY PUSH-BUTTONS
      AN    "MAP_DI".DB91_DBX000_1;
      =     "Db Plc <=> HMI".LINE1.DB100_DBX149_1;
NETWORK
TITLE = CABINET TEMPERATURE
      AN    "MAP_DI".DB91_DBX000_2;
      S     "Db Plc <=> HMI".LINE1.DB100_DBX149_2;
NETWORK
TITLE = SERVICE AUXILIARY 220V TRANSFORMER OVERLOAD
      AN    "MAP_DI".DB91_DBX000_3;
      =     "Db Plc <=> HMI".LINE1.DB100_DBX149_3;
NETWORK
TITLE = CABINET AIR FANS OVERLOAD
      A     "T0";
      AN    "MAP_DI".DB91_DBX000_6;
      =     "Db Plc <=> HMI".LINE1.DB100_DBX149_4;
NETWORK
TITLE = CONTROL DESK FAN OVERLOAD - NOT USED
//NOT USED
      CLR;
      =     "Db Plc <=> HMI".LINE1.DB100_DBX148_2;
NETWORK
TITLE = DRYER OVERLOAD
      A     "T0";
      AN    "MAP_DI".DB91_DBX001_0;
      =     "Db Plc <=> HMI".LINE1.DB100_DBX148_4;
NETWORK
TITLE = AC MOTORS DRIVES FEEDER DC BUS FAULT 
      A     "T0";
      AN    "MAP_DI".DB91_DBX001_2;
      S     "Db Plc <=> HMI".LINE1.DB100_DBX148_1;
NETWORK
TITLE = AC MOTORS DRIVES FEEDER BRAKING RESISTOR
      A     "T0";
      A     "MAP_DO".DB93_DBX000_6;
      AN    "MAP_DI".DB91_DBX001_1;
      L     S5T#3S;
      SD    "T6";
      NOP   0;
      NOP   0;
      NOP   0;
      A     "T6";
      S     "Db Plc <=> HMI".LINE1.DB100_DBX148_5;
NETWORK
TITLE = LINE STOP SERIES PUSH-BUTTON
      A     "T0";
      AN    "M180.1";
      A(;
      ON    "M20.7";
      ON    "M21.0";
      );
      =     "Db Plc <=> HMI".LINE1.DB100_DBX149_5;
NETWORK
TITLE = LINEAR OVERSPEED
      A     "T0";
      A     "M180.1";
      A(;
      L     "Line".DB55_DBD68;
      L     6.200000e+01;
      >=R;
      );
      S     "Db Plc <=> HMI".LINE1.DB100_DBX149_6;
NETWORK
TITLE = 24VDC AUXILIARY FEEDING OVERLOAD
      A     "T0";
      AN    "MAP_DI".DB91_DBX003_1;
      =     "Db Plc <=> HMI".LINE_21.DB100_DBX150_0;
NETWORK
TITLE = 230VAC AUXILIARY FEEDING OVERLOAD
      A     "T0";
      AN    "MAP_DI".DB91_DBX003_2;
      =     "Db Plc <=> HMI".LINE_21.DB100_DBX150_1;
NETWORK
TITLE = AC MOTOR DRIVE  FEEDER FAN OVERLOAD
      A     "T0";
      AN    "MAP_DI".DB91_DBX003_3;
      =     "Db Plc <=> HMI".LINE_21.DB100_DBX150_2;
NETWORK
TITLE = 24VDC PLC INPUT SUPPLY OVERLOAD
      AN    "MAP_DI".DB91_DBX003_4;
      =     "Db Plc <=> HMI".LINE_21.DB100_DBX150_3;
NETWORK
TITLE = 230VAC UPS GENERAL ALARM
      A     "T0";
      A     "MAP_DI".DB91_DBX002_7;
      A     "MAP_DI".DB91_DBX002_5;
      S     "Db Plc <=> HMI".LINE_21.DB100_DBX151_0;
NETWORK
TITLE = 230VAC UPS BATTERY NEARLY LOW
      A     "T0";
      A     "MAP_DI".DB91_DBX003_0;
      =     "Db Plc <=> HMI".LINE_21.DB100_DBX151_1;
NETWORK
TITLE = 230VAC UPS LINE VOLTAGE MISSING - UPS IS OPERATING - NOT USED
//NOT USED
      CLR;
      =     "Db Plc <=> HMI".LINE_21.DB100_DBX151_2;
NETWORK
TITLE = 24VDC UPS MODULE ALARM
      A     "T0";
      AN    "MAP_DI".DB91_DBX000_4;
      S     "Db Plc <=> HMI".LINE_21.DB100_DBX151_3;
NETWORK
TITLE = 24VDC UPS LINE VOLTAGE MISSING - UPS IS OPERATING
      A     "T0";
      AN    "MAP_DI".DB91_DBX000_5;
      =     "Db Plc <=> HMI".LINE_21.DB100_DBX151_4;
NETWORK
TITLE = LINE GENERAL ALARM
      AN    "Db Plc <=> HMI".LINE1.DB100_DBX149_0;
      AN    "Db Plc <=> HMI".LINE1.DB100_DBX149_1;
      AN    "Db Plc <=> HMI".LINE1.DB100_DBX149_2;
      AN    "Db Plc <=> HMI".LINE1.DB100_DBX149_3;
      AN    "Db Plc <=> HMI".LINE1.DB100_DBX149_4;
      AN    "Db Plc <=> HMI".LINE1.DB100_DBX149_5;
      AN    "Db Plc <=> HMI".LINE1.DB100_DBX149_6;
      AN    "Db Plc <=> HMI".LINE1.DB100_DBX148_1;
      AN    "Db Plc <=> HMI".LINE1.DB100_DBX148_2;
      AN    "Db Plc <=> HMI".LINE1.DB100_DBX148_4;
      AN    "Db Plc <=> HMI".LINE1.DB100_DBX148_5;
      AN    "Db Plc <=> HMI".LINE_21.DB100_DBX150_0;
      AN    "Db Plc <=> HMI".LINE_21.DB100_DBX150_1;
      AN    "Db Plc <=> HMI".LINE_21.DB100_DBX150_2;
      AN    "Db Plc <=> HMI".LINE_21.DB100_DBX150_3;
      AN    "Db Plc <=> HMI".LINE_21.DB100_DBX151_0;
      AN    "Db Plc <=> HMI".LINE_21.DB100_DBX151_1;
      AN    "Db Plc <=> HMI".LINE_21.DB100_DBX151_3;
      =     "M197.0";
END_FUNCTION

FUNCTION "Line unit" : VOID	// FC 53
TITLE = LINE UNIT FUNCTION
AUTHOR : Milesi
VERSION : 0.1
BEGIN
NETWORK
TITLE = MASTER CAGE SELECTION 
      AN    "M190.0";
      JC    C006;
      L     "Cage 6".DB30_DBD108;
      T     "Line".DB55_DBD88;
      L     "Cage 6".DB30_DBW14;
      ITD;
      DTR;
      T     "Line".DB55_DBD192;
      JU    END1;
C006: AN    "M188.0";
      JC    C012;
      L     "Cage 12".DB25_DBD108;
      T     "Line".DB55_DBD88;
      L     "Cage 12".DB25_DBW14;
      ITD;
      DTR;
      T     "Line".DB55_DBD192;
      JU    END1;
C012: AN    "M186.0";
      JC    C018;
      L     "Cage 18".DB20_DBD108;
      T     "Line".DB55_DBD88;
      L     "Cage 18".DB20_DBW14;
      ITD;
      DTR;
      T     "Line".DB55_DBD192;
      JU    END1;
C018: AN    "M192.0";
      JC    C024;
      L     "Cage 24".DB15_DBD108;
      T     "Line".DB55_DBD88;
      L     "Cage 24".DB15_DBW14;
      ITD;
      DTR;
      T     "Line".DB55_DBD192;
      JU    END1;
C024: L     6.300000e+02;
      T     "Line".DB55_DBD192;
END1: NOP   0;
NETWORK
TITLE = COPPER-ALLUMINIUM SELECTION
      AN    "M180.1";
      AN    "M20.0";
      A     "Line".HMI_Bit.DB55_DBX1_1;
      S     "M200.1";
      AN    "M180.1";
      AN    "M20.0";
      AN    "Line".HMI_Bit.DB55_DBX1_1;
      R     "M200.1";
      NOP   0;
NETWORK
TITLE = CABLE TYPE SELECTION
// Straight sectoral cable
      AN    "M180.1";
      AN    "M20.0";
      A(;
      L     "Line".DB55_DBW2;
      L     0;
      ==I;
      );
      S     "M200.2";
      R     "M200.3";
      R     "M200.4";
// Preformed sectoral cable
      AN    "M180.1";
      AN    "M20.0";
      A(;
      L     "Line".DB55_DBW2;
      L     1;
      ==I;
      );
      R     "M200.2";
      S     "M200.3";
      R     "M200.4";
// Round cable
      AN    "M180.1";
      AN    "M20.0";
      A(;
      L     "Line".DB55_DBW2;
      L     2;
      ==I;
      );
      R     "M200.2";
      R     "M200.3";
      S     "M200.4";
NETWORK
TITLE = AUXILIARY ON ON-DELAY TIMER
      A     "MAP_DI".DB91_DBX000_0;
      L     S5T#3S;
      SD    "T0";
      NOP   0;
      NOP   0;
      NOP   0;
      NOP   0;
NETWORK
TITLE = BOBBINS DIAMETER CALCULATION SET POINT
      A     "M180.0";
      A(;
      L     "Line".DB55_DBD68;
      L     3.000000e+00;
      >R;
      );
      A     "M200.7";
      AN    "Db Plc <=> HMI".LINE1.DB100_DBX149_7;
      =     "M201.0";
NETWORK
TITLE = BREAKING CONTROL ON-DELAY TIMER
      L     "Line".DB55_DBD136;
      RND;
      ITB;
      L     W#16#2000;
      OW;
      T     "MW264";
NETWORK
TITLE =
      A     "T0";
      A     "M180.0";
      L     "MW264";
      SD    "T1";
      NOP   0;
      NOP   0;
      NOP   0;
      NOP   0;
NETWORK
TITLE = BREAKING CONTROL SET POINT
      A     "M180.0";
      A(;
      L     "Line".DB55_DBD68;
      L     3.000000e+00;
      >R;
      );
      A     "T1";
      =     "M201.2";
NETWORK
TITLE = BRAKES-OIL CONTROL ON-DELAY TIMER
      L     "Line".DB55_DBD140;
      RND;
      ITB;
      L     W#16#2000;
      OW;
      T     "MW266";
NETWORK
TITLE =
      O     "M180.0";
      O     "M180.3";
      O     "M20.6";
      L     "MW266";
      SD    "T2";
      NOP   0;
      NOP   0;
      NOP   0;
      NOP   0;
NETWORK
TITLE = GUARDS BLOWERS OFF-DELAY TIMER
      L     "Line".DB55_DBD144;
      RND;
      ITB;
      L     W#16#2000;
      OW;
      T     "M270";
NETWORK
TITLE =
      A     "M180.1";
      L     "M270";
      SF    "T3";
      NOP   0;
      NOP   0;
      NOP   0;
      NOP   0;
NETWORK
TITLE = DRIVES FEEDER START
      A     "MAP_DI".DB91_DBX000_0;
      AN    "Db Plc <=> HMI".LINE1.DB100_DBX148_1;
      AN    "Db Plc <=> HMI".LINE1.DB100_DBX148_5;
      AN    "M220.0";
      =     "MAP_DO".DB93_DBX000_6;
NETWORK
TITLE = 230AC UPS AUTOMATIC SHUT-DOWN
      AN    "MAP_DI".DB91_DBX002_6;
      =     "MAP_DO".DB93_DBX002_0;
NETWORK
TITLE = ALARMS RESET PILOT LAMP
      AN    "M102.1";
      A     "M1.5";
      =     "MAP_DO".DB93_DBX000_1;
      =     "MAP_DO".DB93_DBX022_4;
      =     "MAP_DO".DB93_DBX032_4;
      =     "MAP_DO".DB93_DBX042_4;
      =     "MAP_DO".DB93_DBX052_4;
END_FUNCTION

FUNCTION "Run consent" : VOID	// FC 54
TITLE = RUN CONSENT FUNCTION
AUTHOR : Milesi
VERSION : 0.1
BEGIN
NETWORK
TITLE = RUN CONSENT
      A     "M195.0";
      A     "M195.1";
      A     "M197.3";
      A     "M196.1";
      A     "M196.2";
      A     "M195.7";
      A     "M196.0";
      A     "M195.5";
      A     "M195.6";
      A     "M195.3";
      A     "M195.4";
      A     "M196.3";
      A     "M197.0";
      A     "M196.7";
      =     "M102.0";
NETWORK
TITLE = RUN CONSENT WITH TAKE-UP ON
      A     "M102.0";
      AN    "Db Plc <=> HMI".TAKE_UP_1.DB100_DBX106_1;
      =     "M102.1";
NETWORK
TITLE = READY TO RUN
      A     "M102.1";
      AN    "M180.1";
      =     "Db Plc <=> HMI".LINE1.DB100_DBX148_7;
END_FUNCTION

FUNCTION "Line jog - line run" : VOID	// FC 55
TITLE = LINE JOG-LINE RUN FUNCTION
AUTHOR : Milesi
VERSION : 0.1
VAR_TEMP
  T4_time : S5TIME ;	//T1 BCD time set from MP
END_VAR
BEGIN
NETWORK
TITLE = LINE RUN REQUEST
      A(;
      O     "MAP_DI".DB91_DBX002_1;
      O     "MAP_DI".DB91_DBX002_2;
      O     "M20.3";
      O     "M20.2";
      O     "M20.4";
      );
      A     "MAP_DI".DB91_DBX000_1;
      A     "M20.7";
      A     "M21.0";
      =     "M178.0";
NETWORK
TITLE = LINE RUN ON-DELAY TIMER
      L     "Line".DB55_DBD132;
      RND;
      ITB;
      L     W#16#2000;
      OW;
      T     "MW268";
NETWORK
TITLE =
      A(;
      A     "M178.0";
      L     "MW268";
      SD    "T4";
      NOP   0;
      NOP   0;
      NOP   0;
      A     "T4";
      );
      AN    "T4";
      AN    "M180.1";
      A     "M102.1";
      A     "M1.4";
      =     "MAP_DO".DB93_DBX000_3;
NETWORK
TITLE = LINE RUN SIREN
      A     "M178.0";
      AN    "T4";
      AN    "M180.1";
      A     "M102.1";
      A     "M1.4";
      =     "MAP_DO".DB93_DBX000_3;
NETWORK
TITLE = CAGE 6 AC MOTOR JOG FOR LOADING STROKE
      A     "T41";
      =     "M190.4";
NETWORK
TITLE = CAGE 12 AC MOTOR JOG FOR LOADING STROKE
      A     "T31";
      =     "M188.4";
NETWORK
TITLE = CAGE 18 AC MOTOR JOG FOR LOADING STROKE
      A     "T21";
      =     "M186.4";
NETWORK
TITLE = CAGE 18 AC MOTOR JOG FOR LOADING STROKE
      A     "T15";
      =     "M192.4";
NETWORK
TITLE = LINE JOG
      A(;
      O     "MAP_DI".DB91_DBX002_2;
      O     "M20.4";
      O     "M20.2";
      );
      A     "T4";
      AN    "M180.0";
      A     "M102.1";
      A     "MAP_DI".DB91_DBX000_1;
      A     "M20.7";
      A     "M21.0";
      AN    "M220.0";
      =     "M180.3";
NETWORK
TITLE = LINE RUN WITHOUT ZERO SPEED
      A(;
      A     "MAP_DI".DB91_DBX002_1;
      A     "T4";
      AN    "Drives --> Plc".CAPSTAN_STATUS_W1.DB1_DBX80_2;
      O;
      A     "M180.0";
      A(;
      O     "Drives --> Plc".CAPSTAN_STATUS_W1.DB1_DBX80_2;
      ON    "M220.0";
      );
      );
      AN    "M180.3";
      A     "M102.1";
      A     "MAP_DI".DB91_DBX000_1;
      A     "M20.7";
      A     "M21.0";
      =     "M180.0";
NETWORK
TITLE = LINE RUN WITH ZERO SPEED
      A     "M180.1";
      A     "Drives --> Plc".CAPSTAN_STATUS_W1.DB1_DBX80_2;
      O     "M180.0";
      O     "M180.3";
      =     "M180.1";
NETWORK
TITLE = LINE RUN PILOT LAMP
      O     "M180.0";
      O     "M180.3";
      O;
      A     "M180.1";
      A     "M1.3";
      =     "MAP_DO".DB93_DBX000_0;
NETWORK
TITLE = MACHINE RUNNING
      A     "M180.1";
      =     "Db Plc <=> HMI".LINE1.DB100_DBX148_6;
NETWORK
TITLE = QUICK STOP
      A(;
      O     "Db Plc <=> HMI".PROFIBUS.DB100_DBX100_0;
      O     "Db Plc <=> HMI".PROFIBUS.DB100_DBX100_1;
      O     "Db Plc <=> HMI".PROFIBUS.DB100_DBX100_2;
      O     "Db Plc <=> HMI".PROFIBUS.DB100_DBX100_3;
      O     "Db Plc <=> HMI".PROFIBUS.DB100_DBX100_4;
      O     "Db Plc <=> HMI".PROFIBUS.DB100_DBX100_5;
      O     "Db Plc <=> HMI".PROFIBUS.DB100_DBX100_6;
      O     "Db Plc <=> HMI".PROFIBUS.DB100_DBX100_7;
      O     "Db Plc <=> HMI".PROFIBUS.DB100_DBX101_0;
      O     "Db Plc <=> HMI".PROFIBUS.DB100_DBX101_1;
      O     "Db Plc <=> HMI".PROFIBUS.DB100_DBX101_2;
      O     "Db Plc <=> HMI".PROFIBUS.DB100_DBX101_5;
      O     "Db Plc <=> HMI".PROFIBUS.DB100_DBX101_6;
      O     "Db Plc <=> HMI".PROFIBUS.DB100_DBX101_7;
      O     "Db Plc <=> HMI".PROFIBUS_1.DB100_DBX103_0;
      O     "Db Plc <=> HMI".PROFIBUS_1.DB100_DBX103_1;
      O     "Db Plc <=> HMI".PROFIBUS_1.DB100_DBX103_2;
      O     "Db Plc <=> HMI".TRAVERSE.DB100_DBX105_3;
      O     "Db Plc <=> HMI".TAKE_UP_1.DB100_DBX107_6;
      O     "Db Plc <=> HMI".CAPSTAN.DB100_DBX109_6;
      O     "Db Plc <=> HMI".CAGE24_3.DB100_DBX117_06;
      O     "Db Plc <=> HMI".CAGE24_4.DB100_DBX118_05;
      O     "Db Plc <=> HMI".CAGE24_4.DB100_DBX119_07;
      O     "Db Plc <=> HMI".CAGE18_3.DB100_DBX125_06;
      O     "Db Plc <=> HMI".CAGE18_4.DB100_DBX126_05;
      O     "Db Plc <=> HMI".CAGE18_4.DB100_DBX127_07;
      O     "Db Plc <=> HMI".Cage12_3.DB100_DBX133_06;
      O     "Db Plc <=> HMI".Cage12_4.DB100_DBX134_05;
      O     "Db Plc <=> HMI".Cage12_4.DB100_DBX135_07;
      O     "Db Plc <=> HMI".Cage6_3.DB100_DBX141_6;
      O     "Db Plc <=> HMI".Cage6_4.DB100_DBX142_5;
      O     "Db Plc <=> HMI".PAY_OFF_UNIT1.DB100_DBX144_2;
      O     "Db Plc <=> HMI".PAY_OFF_UNIT1.DB100_DBX145_6;
      O     "M178.5";
      O     "M178.6";
      O     "M178.7";
      O     "M179.0";
      ON    "MAP_DI".DB91_DBX000_1;
      );
      S     "M179.1";
      AN    "M180.1";
      R     "M179.1";
      NOP   0;
END_FUNCTION

FUNCTION "Line reference" : VOID	// FC 56
TITLE = LINE REFERENCE FUNCTION
AUTHOR : Milesi
VERSION : 0.1
BEGIN
NETWORK
TITLE = MAXIMUM LINEAR SPEED FROM HMI
      A(;
      L     "Line".DB55_DBD28;
      L     "Line".DB55_DBD32;
      >R;
      );
      JNB   _001;
      L     "Line".DB55_DBD32;
      T     "Line".DB55_DBD28;
_001: NOP   0;
NETWORK
TITLE = MAXIMUM LINEAR SPEED SET TO HMI
      A(;
      L     "Line".DB55_DBD28;
      L     "Line".DB55_DBD40;
      >R;
      );
      JNB   _003;
      L     "Line".DB55_DBD40;
      T     "Line".DB55_DBD28;
_003: NOP   0;
NETWORK
TITLE = LINE RUN SPEED REFERENCE
      L     "Line".DB55_DBD28;
      T     "Line".DB55_DBD48;
      NOP   0;
NETWORK
TITLE = LINE JOG SPEED REFERENCE
      A     "M180.3";
      JNB   _007;
      L     "Line".DB55_DBD36;
      T     "Line".DB55_DBD48;
_007: NOP   0;
NETWORK
TITLE = MAX LINEAR SPEED TO START
      A(;
      L     "Cage 6".DB30_DBD120;
      L     "Cage 12".DB25_DBD120;
      <=R;
      );
      A(;
      L     "Cage 6".DB30_DBD120;
      L     "Cage 18".DB20_DBD120;
      <=R;
      );
      A(;
      L     "Cage 6".DB30_DBD120;
      L     "Cage 24".DB15_DBD120;
      <=R;
      );
      A     "M190.0";
      JNB   _030;
      L     "Cage 6".DB30_DBD120;
      T     "Line".DB55_DBD72;
      JU    END;
_030: A(;
      L     "Cage 12".DB25_DBD120;
      L     "Cage 6".DB30_DBD120;
      <=R;
      );
      A(;
      L     "Cage 12".DB25_DBD120;
      L     "Cage 18".DB20_DBD120;
      <=R;
      );
      A(;
      L     "Cage 12".DB25_DBD120;
      L     "Cage 24".DB15_DBD120;
      <=R;
      );
      A     "M188.0";
      JNB   _031;
      L     "Cage 12".DB25_DBD120;
      T     "Line".DB55_DBD72;
      JU    END;
_031: A(;
      L     "Cage 18".DB20_DBD120;
      L     "Cage 6".DB30_DBD120;
      <=R;
      );
      A(;
      L     "Cage 18".DB20_DBD120;
      L     "Cage 12".DB25_DBD120;
      <=R;
      );
      A(;
      L     "Cage 18".DB20_DBD120;
      L     "Cage 24".DB15_DBD120;
      <=R;
      );
      A     "M186.0";
      JNB   _032;
      L     "Cage 18".DB20_DBD120;
      T     "Line".DB55_DBD72;
      JU    END;
_032: A(;
      L     "Cage 24".DB15_DBD120;
      L     "Cage 6".DB30_DBD120;
      <=R;
      );
      A(;
      L     "Cage 24".DB15_DBD120;
      L     "Cage 12".DB25_DBD120;
      <=R;
      );
      A(;
      L     "Cage 24".DB15_DBD120;
      L     "Cage 18".DB20_DBD120;
      <=R;
      );
      A     "M192.0";
      JNB   END;
      L     "Cage 24".DB15_DBD120;
      T     "Line".DB55_DBD72;
      JU    END;
END:  A     "M190.0";
      O     "M188.0";
      O     "M186.0";
      O     "M192.0";
      JC    J00;
      L     6.000000e+01;
      T     "Line".DB55_DBD72;
J00:  NOP   0;
NETWORK
TITLE = MAX LINEAR SPEED
      A(;
      L     "Cage 6".DB30_DBD96;
      L     "Cage 12".DB25_DBD96;
      <=R;
      );
      A(;
      L     "Cage 6".DB30_DBD96;
      L     "Cage 18".DB20_DBD96;
      <=R;
      );
      A(;
      L     "Cage 6".DB30_DBD96;
      L     "Cage 24".DB15_DBD96;
      <=R;
      );
      A     "M190.0";
      JNB   _060;
      L     "Cage 6".DB30_DBD96;
      JU    END1;
_060: A(;
      L     "Cage 12".DB25_DBD96;
      L     "Cage 6".DB30_DBD96;
      <=R;
      );
      A(;
      L     "Cage 12".DB25_DBD96;
      L     "Cage 18".DB20_DBD96;
      <=R;
      );
      A(;
      L     "Cage 12".DB25_DBD96;
      L     "Cage 24".DB15_DBD96;
      <=R;
      );
      A     "M188.0";
      JNB   _061;
      L     "Cage 12".DB25_DBD96;
      JU    END1;
_061: A(;
      L     "Cage 18".DB20_DBD96;
      L     "Cage 6".DB30_DBD96;
      <=R;
      );
      A(;
      L     "Cage 18".DB20_DBD96;
      L     "Cage 12".DB25_DBD96;
      <=R;
      );
      A(;
      L     "Cage 18".DB20_DBD96;
      L     "Cage 24".DB15_DBD96;
      <=R;
      );
      A     "M186.0";
      JNB   _062;
      L     "Cage 18".DB20_DBD96;
      JU    END1;
_062: A(;
      L     "Cage 24".DB15_DBD96;
      L     "Cage 6".DB30_DBD96;
      <=R;
      );
      A(;
      L     "Cage 24".DB15_DBD96;
      L     "Cage 12".DB25_DBD96;
      <=R;
      );
      A(;
      L     "Cage 24".DB15_DBD96;
      L     "Cage 18".DB20_DBD96;
      <=R;
      );
      A     "M192.0";
      JNB   END1;
      L     "Cage 24".DB15_DBD96;
      JU    END1;
END1: A     "M200.2";
      JNB   END2;
      L     4.000000e+01;
      <=R;
      JNB   END2;
      TAK;
      JU    Fend;
END2: A     "M200.3";
      JNB   END3;
      L     4.000000e+01;
      <=R;
      JNB   END3;
      TAK;
      JU    Fend;
END3: A     "M200.4";
      JNB   Fend;
      L     6.000000e+01;
      <=R;
      JNB   Fend;
      TAK;
Fend: T     "Line".DB55_DBD40;
NETWORK
TITLE = LINE SPEED TO START + LINE INCREASE RPM
      L     "Line".DB55_DBD72;
      L     "Line".DB55_DBD76;
      +R;
      T     "Line".DB55_DBD80;
NETWORK
TITLE = LINE SPEED LIMIT CONTROL AND ADJUSTMENT FOR RAMP
      A(;
      L     "Line".DB55_DBD48;
      L     "Line".DB55_DBD80;
      >=R;
      );
      JNB   OPER;
      L     1.666667e+02;
      *R;
      T     "Line".DB55_DBD84;
      JU    OUT;
OPER: L     "Line".DB55_DBD48;
      L     1.666667e+02;
      *R;
      T     "Line".DB55_DBD84;
OUT:  NOP   0;
NETWORK
TITLE = MAXIMUM RAMP INPUT
      A(;
      L     1.000000e+04;
      L     "Line".DB55_DBD84;
      <R;
      );
      JNB   _00b;
      L     1.000000e+04;
      T     "Line".DB55_DBD84;
_00b: NOP   0;
NETWORK
TITLE = LINE QUICK STOP RAMP DOWN TIME
      AN    "MAP_DI".DB91_DBX000_1;
      JC    BL4;
      L     1.200000e+01;
      T     "Line".DB55_DBD64;
BL4:  NOP   0;
NETWORK
TITLE = LINE EMERGENCY STOP RAMP DOWN TIME
      A     "MAP_DI".DB91_DBX000_1;
      JC    BL5;
      L     7.000000e+00;
      T     "Line".DB55_DBD64;
BL5:  NOP   0;
NETWORK
TITLE = RAMP ENABLE
      O     "M180.0";
      O     "M180.3";
      =     "M201.1";
NETWORK
TITLE = RAMP
      CALL  "Ramp" (
           INPUT_10000              := "Line".DB55_DBD84,
           UP_DOWN_sec              := "Line".DB55_DBD44,
           NORMAL_STOP_sec          := 2.000000e+01,
           QUICK_STOP_sec           := "Line".DB55_DBD64,
           HOLD_LAMP                := "MAP_DO".DB93_DBX000_2,
           FIXED_RAMP               := "M200.7",
           RAMP_ENABLE              := "M201.1",
           SLOW_DOWN                := "Db Plc <=> HMI".LINE1.DB100_DBX149_7,
           QUICK_STOP               := "M179.1",
           HOLD                     := "MAP_DI".DB91_DBX002_4,
           HOLD_FLAG                := "M12.0",
           HOLD_FLAG_1              := "M12.1",
           OUTPUT_REAL_10000        := "Line".DB55_DBD96,
           OUTPUT_DINT_10000        := "Line".DB55_DBD100,
           OUTPUT_REAL_100          := "Line".DB55_DBD104,
           MEM_FLAG1                := "M12.2",
           MEM_FLAG2                := "M12.3",
           MEM_FLAG3                := "M12.4",
           MEM_FLAG4                := "M12.5",
           MEM_FLAG5                := "M12.6",
           MEM_FLAG6                := "M12.7");
NETWORK
TITLE = RAMP OUTPUT RESET
      A     "M180.1";
      JC    _004;
      L     0.000000e+00;
      T     "Line".DB55_DBD96;
      T     "Line".DB55_DBD100;
      T     "Line".DB55_DBD104;
_004: NOP   0;
NETWORK
TITLE = LINE LINEAR SPEED REFERENCE
      L     "Line".DB55_DBD96;
      L     1.000000e+04;
      /R;
      L     6.000000e+01;
      *R;
      T     "Line".DB55_DBD60;
NETWORK
TITLE = CAGE 6 LOADING LINEAR SPEED REFERENCE
      A     "M180.4";
      A     "M190.0";
      JNB   _105;
      L     "Cage 6".DB30_DBD24;
      L     "Cage 6".DB30_DBD108;
      *R;
      L     1.000000e+00;
      *R;
      L     1.000000e+03;
      /R;
      T     "Line".DB55_DBD60;
_105: NOP   0;
NETWORK
TITLE = CAGE 12 LOADING LINEAR SPEED REFERENCE
      A     "M180.5";
      A     "M188.0";
      JNB   _005;
      L     "Cage 12".DB25_DBD24;
      L     "Cage 12".DB25_DBD108;
      *R;
      L     1.000000e+00;
      *R;
      L     1.000000e+03;
      /R;
      T     "Line".DB55_DBD60;
_005: NOP   0;
NETWORK
TITLE = CAGE 18 LOADING LINEAR SPEED REFERENCE
      A     "M180.6";
      A     "M186.0";
      JNB   _006;
      L     "Cage 18".DB20_DBD24;
      L     "Cage 18".DB20_DBD108;
      *R;
      L     1.000000e+00;
      *R;
      L     1.000000e+03;
      /R;
      T     "Line".DB55_DBD60;
_006: NOP   0;
NETWORK
TITLE = CAGE 24 LOADING LINEAR SPEED REFERENCE
      A     "M180.7";
      A     "M192.0";
      JNB   _107;
      L     "Cage 24".DB15_DBD24;
      L     "Cage 24".DB15_DBD108;
      *R;
      L     1.000000e+00;
      *R;
      L     1.000000e+03;
      /R;
      T     "Line".DB55_DBD60;
_107: NOP   0;
NETWORK
TITLE = MISSING POWER SUPPLY LINEAR SPEED REFERENCE
      A     "M202.0";
      A     "M220.0";
      JCN   mas1;
      L     "Cage 6".DB30_DBD24;
      L     "Cage 6".DB30_DBD108;
      *R;
      L     1.000000e+03;
      /R;
      JU    rif;
mas1: A     "M202.1";
      A     "M220.0";
      JCN   mas2;
      L     "Cage 12".DB25_DBD24;
      L     "Cage 12".DB25_DBD108;
      *R;
      L     1.000000e+03;
      /R;
      JU    rif;
mas2: A     "M202.2";
      A     "M220.0";
      JCN   mas3;
      L     "Cage 18".DB20_DBD24;
      L     "Cage 18".DB20_DBD108;
      *R;
      L     1.000000e+03;
      /R;
      JU    rif;
mas3: A     "M202.3";
      A     "M220.0";
      JCN   mas4;
      L     "Cage 24".DB15_DBD24;
      L     "Cage 24".DB15_DBD108;
      *R;
      L     1.000000e+03;
      /R;
mas4: NOP   0;
rif:  T     "Line".DB55_DBD60;
END_FUNCTION

FUNCTION "Linear speed" : VOID	// FC 57
TITLE = LINEAR SPEED FUNCTION
AUTHOR : Milesi
VERSION : 0.1
VAR_TEMP
  Aux : REAL ;
END_VAR
BEGIN
NETWORK
TITLE = LINEAR SPEED CALCULATION ENABLE
      O     "M180.1";
      O     "M21.3";
      O     "M184.2";
      =     "M179.6";
NETWORK
TITLE = CAPSTAN LINEAR SPEED CONVERSION
      L     "Drives --> Plc".DB1_DBW86;
      ITD;
      DTR;
      T     "Capstan".DB9_DBD68;
NETWORK
TITLE = CAPSTAN LINEAR SPEED CALCULATION
      CALL  "Capstan linear speed" (
           Enable                   := "M179.6",
           Capstan_pulley_diameter  := 2.500000e+03,
           Cable_diameter           := "Line".DB55_DBD56,
           Input_speed              := "Capstan".DB9_DBD68,
           Input_speed_resolution   := 1.638400e+04,
           Max_line_speed           := 6.000000e+01,
           K_filter                 := 1.000000e+00,
           Added_value              := "Capstan".DB9_DBD60,
           Counter_increase         := "Capstan".DB9_DBD64,
           Filtered_linear_speed    := "Line".DB55_DBD68);
END_FUNCTION

FUNCTION "Missing power supply" : VOID	// FC 59
TITLE = MISSING POWER SUPPLY FUNCTION
AUTHOR : Milesi
VERSION : 0.1
VAR_TEMP
  Cage6_theoric_rpm : REAL ;
  Cage12_theoric_rpm : REAL ;
  Cage18_theoric_rpm : REAL ;
  Cage24_theoric_rpm : REAL ;
END_VAR
BEGIN
NETWORK
TITLE = CAGE 6 MASTER OF MISSING POWER SUPPLY
      A     "M190.0";
      AN    "M188.0";
      AN    "M186.0";
      AN    "M192.0";
      AN    "M180.1";
      S     "M202.0";
      R     "M202.1";
      R     "M202.2";
      R     "M202.3";
NETWORK
TITLE = CAGE 12 MASTER OF MISSING POWER SUPPLY
      A     "M188.0";
      AN    "M186.0";
      AN    "M192.0";
      AN    "M180.1";
      R     "M202.0";
      S     "M202.1";
      R     "M202.2";
      R     "M202.3";
NETWORK
TITLE = CAGE 18 MASTER OF MISSING POWER SUPPLY
      A     "M186.0";
      AN    "M192.0";
      AN    "M180.1";
      R     "M202.0";
      R     "M202.1";
      S     "M202.2";
      R     "M202.3";
NETWORK
TITLE = CAGE 24 MASTER OF MISSING POWER SUPPLY
      A     "M192.0";
      AN    "M180.1";
      R     "M202.0";
      R     "M202.1";
      R     "M202.2";
      S     "M202.3";
NETWORK
TITLE = RESET MASTER OF MISSING SUPPLY RAMP DOWN 
      AN    "M190.0";
      AN    "M188.0";
      AN    "M186.0";
      AN    "M192.0";
      R     "M202.0";
      R     "M202.1";
      R     "M202.2";
      R     "M202.3";
NETWORK
TITLE = CAGE 6 KINETIC BUFFERING THRESHOLD
      A     "M202.0";
      JCN   KIB1;
      L     85;
      T     "MW292";
      L     1;
      T     "MW298";
      JU    KIBE;
KIB1: L     65;
      T     "MW292";
      L     0;
      T     "MW298";
KIBE: NOP   0;
NETWORK
TITLE = CAGE 12 KINETIC BUFFERING THRESHOLD
      A     "M202.1";
      JCN   KIB2;
      L     85;
      T     "MW290";
      L     1;
      T     "MW296";
      JU    KIBR;
KIB2: L     65;
      T     "MW290";
      L     0;
      T     "MW296";
KIBR: NOP   0;
NETWORK
TITLE = CAGE 18 KINETIC BUFFERING THRESHOLD
      A     "M202.2";
      JCN   KIB3;
      L     85;
      T     "MW288";
      L     1;
      T     "MW294";
      JU    KIBT;
KIB3: L     65;
      T     "MW288";
      L     0;
      T     "MW294";
KIBT: NOP   0;
NETWORK
TITLE = CAGE 24 KINETIC BUFFERING THRESHOLD
      A     "M202.3";
      JCN   KIB4;
      L     85;
      T     "MW284";
      L     1;
      T     "MW286";
      JU    KIBU;
KIB4: L     65;
      T     "MW284";
      L     0;
      T     "MW286";
KIBU: NOP   0;
NETWORK
TITLE = MISSING POWER SUPPLY START
      A(;
      O     "Drives --> Plc".CAGE_24_STATUS_W1.DB1_DBX160_7;
      O     "Drives --> Plc".CAGE_18_STATUS_W1.DB1_DBX240_7;
      O     "Drives --> Plc".CAGE_12_PREF_STATUS_W1.DB1_DBX280_7;
      O     "Drives --> Plc".CAGE_6_STATUS_W1.DB1_DBX360_7;
      );
      A     "MAP_DI".DB91_DBX000_1;
      A     "M180.1";
      S     "M220.0";
      A     "M30.1";
      R     "M220.0";
      NOP   0;
END_FUNCTION

